ABB RobotStudio station: Laboratorio_simula.rspag

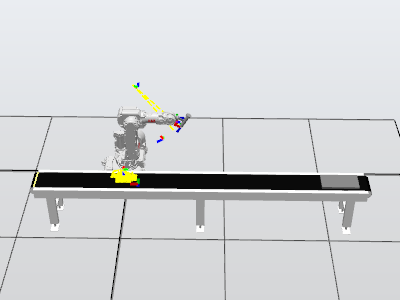
--- station ---
Station Project2 (saved by RobotStudio 25.3.11371.0)
Controller IRB140_6_81
  mechanical unit ROB_1: IRB140_6_81_C_03, 6 joints, base frame (0, 0, 0) mm
Layout (positions relative to the parent item):
  - IRB140_6_81_C_03 [mechanism, from %ABB.RobotStudio.Models.IRB140%\IRB140_6_81_C_G_03.rslib] at (0, 0, 0) mm; joint values [0, 0, 0, 0, 0, 0] (rad or m)
  - Soporte_final [mechanism] at (515, 0, 712) mm, rotated rx 0 ry 90 rz 0 deg
      TCP Soporte_final at (-0.03, 41.69, 114.81) mm, rotated rx 0 ry 30 rz -90 deg
      links: Soporte_7
  - Part_1 [part] at (-100, -130, -23) mm, size 280 x 180 x 80 mm
  - Rutina_Banda [smart component]
      signals: DI Activar_banda
      connections:
        Rutina_Banda.DI_01 -> PhysicsControl.SurfaceVelocityEnabled
        LineSensor_2.SensorOut -> Source.Execute
        Rutina_Banda.Activar_banda -> PhysicsControl.SurfaceVelocityEnabled
    - PhysicsControl [smart component, from Components\PhysicsControl.rslib]
        properties: Object=Belt Conveyor; Behavior=1; SurfaceVelocity=0.2
    - Belt Conveyor [part], size 3227.3 x 408.1 x 489.7 mm
    - Part_2 [part] at (2075.83, -708.5, 486.6) mm, size 350 x 180 x 20 mm
    - Source [smart component, from Components\Source.rslib]
        properties: Source=Part_2; Copy=(none); Parent=(none); Position=[2.079365 -0.71 0.517]; Orientation=[0 0 0]; Transient=true; PhysicsBehavior=-1
    - LineSensor_2 [smart component, from Components\LineSensor.rslib]
        properties: Start=[-0.8 -0.82 0.487]; End=[-0.8 -0.6 0.487]; Length=0.22; Radius=0.00152284263959391; Tag=(none); SenseMultiple=false; SensedPart=(none); SensedPoint=[0 0 0]
      - _sensorPart_ [part], size 3 x 220 x 3 mm
Attachment: Soporte_final is attached to IRB140_6_81_C_03 / Link6
Station logic (signal -> signal, property => property):
  IRB140_6_81.Conveyor_INV -> Rutina_Banda.Activar_banda

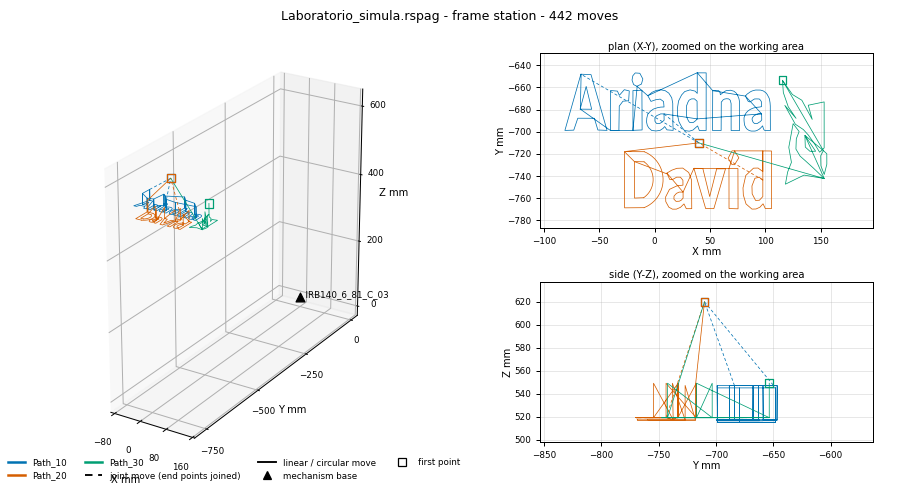
[picture p0: tool path of Laboratorio_simula.rspag in frame station, 442 of 446 moves have a stored position in this frame; points joined in program order, loops and branches not executed]
--- Controller Data/IRB140_6_81/RAPID/TASK1/PROGMOD/CalibData.mod ---
MODULE CalibData
ENDMODULE

--- Controller Data/IRB140_6_81/RAPID/TASK1/PROGMOD/Module3.mod ---
MODULE Module3
    CONST robtarget Target_200:=[[246.278,151.897,-25],[0.707106781,0,0,0.707106781],[-1,0,-1,1],[9E+09,9E+09,9E+09,9E+09,9E+09,9E+09]];
    CONST robtarget Target_210:=[[246.513,151.995,5],[0.707106781,0,0,0.707106781],[-1,0,-1,1],[9E+09,9E+09,9E+09,9E+09,9E+09,9E+09]];
    CONST robtarget Target_220:=[[237.364,151.636,5],[0.707106781,0,0,0.707106781],[-1,0,-1,1],[9E+09,9E+09,9E+09,9E+09,9E+09,9E+09]];
    CONST robtarget Target_230:=[[222.871,101.286,5],[0.707106781,0,0,0.707106781],[-1,0,-1,1],[9E+09,9E+09,9E+09,9E+09,9E+09,9E+09]];
    CONST robtarget Target_240:=[[231.165,101.624,5],[0.707106781,0,0,0.707106781],[-1,0,-1,1],[9E+09,9E+09,9E+09,9E+09,9E+09,9E+09]];
    CONST robtarget Target_250:=[[234.333,112.207,5],[0.707106781,0,0,0.707106781],[-1,0,-1,1],[9E+09,9E+09,9E+09,9E+09,9E+09,9E+09]];
    CONST robtarget Target_260:=[[249.288,112.26,5],[0.707106781,0,0,0.707106781],[-1,0,-1,1],[9E+09,9E+09,9E+09,9E+09,9E+09,9E+09]];
    CONST robtarget Target_270:=[[252.931,101.499,5],[0.707106781,0,0,0.707106781],[-1,0,-1,1],[9E+09,9E+09,9E+09,9E+09,9E+09,9E+09]];
    CONST robtarget Target_280:=[[260.918,101.25,5],[0.707106781,0,0,0.707106781],[-1,0,-1,1],[9E+09,9E+09,9E+09,9E+09,9E+09,9E+09]];
    CONST robtarget Target_290:=[[246.984,120.449,-25],[0.707106781,0,0,0.707106781],[-1,0,-1,1],[9E+09,9E+09,9E+09,9E+09,9E+09,9E+09]];
    CONST robtarget Target_300:=[[247.166,120.45,5],[0.707106781,0,0,0.707106781],[-1,0,-1,1],[9E+09,9E+09,9E+09,9E+09,9E+09,9E+09]];
    CONST robtarget Target_310:=[[236.764,120.36,5],[0.707106781,0,0,0.707106781],[-1,0,-1,1],[9E+09,9E+09,9E+09,9E+09,9E+09,9E+09]];
    CONST robtarget Target_320:=[[241.731,140.965,5],[0.707106781,0,0,0.707106781],[-1,0,-1,1],[9E+09,9E+09,9E+09,9E+09,9E+09,9E+09]];
    CONST robtarget Target_330:=[[219.929,101.246,-25],[0.707106781,0,0,0.707106781],[-1,0,-1,1],[9E+09,9E+09,9E+09,9E+09,9E+09,9E+09]];
    CONST robtarget Target_340:=[[219.745,101.297,5],[0.707106781,0,0,0.707106781],[-1,0,-1,1],[9E+09,9E+09,9E+09,9E+09,9E+09,9E+09]];
    CONST robtarget Target_350:=[[212.197,101.132,5],[0.707106781,0,0,0.707106781],[-1,0,-1,1],[9E+09,9E+09,9E+09,9E+09,9E+09,9E+09]];
    CONST robtarget Target_360:=[[211.858,123.214,5],[0.707106781,0,0,0.707106781],[-1,0,-1,1],[9E+09,9E+09,9E+09,9E+09,9E+09,9E+09]];
    CONST robtarget Target_370:=[[208.528,127.633,5],[0.707106781,0,0,0.707106781],[-1,0,-1,1],[9E+09,9E+09,9E+09,9E+09,9E+09,9E+09]];
    CONST robtarget Target_380:=[[203.388,128.012,5],[0.707106781,0,0,0.707106781],[-1,0,-1,1],[9E+09,9E+09,9E+09,9E+09,9E+09,9E+09]];
    CONST robtarget Target_390:=[[202.821,136.911,5],[0.707106781,0,0,0.707106781],[-1,0,-1,1],[9E+09,9E+09,9E+09,9E+09,9E+09,9E+09]];
    CONST robtarget Target_400:=[[207.318,137.995,5],[0.707106781,0,0,0.707106781],[-1,0,-1,1],[9E+09,9E+09,9E+09,9E+09,9E+09,9E+09]];
    CONST robtarget Target_410:=[[211.798,132.906,5],[0.707106781,0,0,0.707106781],[-1,0,-1,1],[9E+09,9E+09,9E+09,9E+09,9E+09,9E+09]];
    CONST robtarget Target_420:=[[213.511,136.735,5],[0.707106781,0,0,0.707106781],[-1,0,-1,1],[9E+09,9E+09,9E+09,9E+09,9E+09,9E+09]];
    CONST robtarget Target_430:=[[219.776,137.262,5],[0.707106781,0,0,0.707106781],[-1,0,-1,1],[9E+09,9E+09,9E+09,9E+09,9E+09,9E+09]];
    CONST robtarget Target_440:=[[219.929,116.68,5],[0.707106781,0,0,0.707106781],[-1,0,-1,1],[9E+09,9E+09,9E+09,9E+09,9E+09,9E+09]];
    CONST robtarget Target_450:=[[199.531,101.071,-27],[0.707106781,0,0,0.707106781],[-1,0,-1,1],[9E+09,9E+09,9E+09,9E+09,9E+09,9E+09]];
    CONST robtarget Target_460:=[[199.496,101.319,3],[0.707106781,0,0,0.707106781],[-1,0,-1,1],[9E+09,9E+09,9E+09,9E+09,9E+09,9E+09]];
    CONST robtarget Target_470:=[[199.502,137.231,3],[0.707106781,0,0,0.707106781],[-1,0,-1,1],[9E+09,9E+09,9E+09,9E+09,9E+09,9E+09]];
    CONST robtarget Target_480:=[[191.425,137.513,3],[0.707106781,0,0,0.707106781],[-1,0,-1,1],[9E+09,9E+09,9E+09,9E+09,9E+09,9E+09]];
    CONST robtarget Target_490:=[[191.227,101.671,3],[0.707106781,0,0,0.707106781],[-1,0,-1,1],[9E+09,9E+09,9E+09,9E+09,9E+09,9E+09]];
    CONST robtarget Target_500:=[[195.697,140.971,-27],[0.707106781,0,0,0.707106781],[-1,0,-1,1],[9E+09,9E+09,9E+09,9E+09,9E+09,9E+09]];
    CONST robtarget Target_510:=[[195.891,141.123,3],[0.707106781,0,0,0.707106781],[-1,0,-1,1],[9E+09,9E+09,9E+09,9E+09,9E+09,9E+09]];
    CONST robtarget Target_520:=[[191.844,143.083,3],[0.707106781,0,0,0.707106781],[-1,0,-1,1],[9E+09,9E+09,9E+09,9E+09,9E+09,9E+09]];
    CONST robtarget Target_530:=[[190.566,147.695,3],[0.707106781,0,0,0.707106781],[-1,0,-1,1],[9E+09,9E+09,9E+09,9E+09,9E+09,9E+09]];
    CONST robtarget Target_540:=[[193.297,152.839,3],[0.707106781,0,0,0.707106781],[-1,0,-1,1],[9E+09,9E+09,9E+09,9E+09,9E+09,9E+09]];
    CONST robtarget Target_550:=[[197.437,153.127,3],[0.707106781,0,0,0.707106781],[-1,0,-1,1],[9E+09,9E+09,9E+09,9E+09,9E+09,9E+09]];
    CONST robtarget Target_560:=[[199.597,150.616,3],[0.707106781,0,0,0.707106781],[-1,0,-1,1],[9E+09,9E+09,9E+09,9E+09,9E+09,9E+09]];
    CONST robtarget Target_570:=[[200.339,146.707,3],[0.707106781,0,0,0.707106781],[-1,0,-1,1],[9E+09,9E+09,9E+09,9E+09,9E+09,9E+09]];
    CONST robtarget Target_580:=[[198.927,142.651,3],[0.707106781,0,0,0.707106781],[-1,0,-1,1],[9E+09,9E+09,9E+09,9E+09,9E+09,9E+09]];
    CONST robtarget Target_590:=[[196.108,141.187,3],[0.707106781,0,0,0.707106781],[-1,0,-1,1],[9E+09,9E+09,9E+09,9E+09,9E+09,9E+09]];
    CONST robtarget Target_600:=[[185.991,132.618,-27],[0.707106781,0,0,0.707106781],[-1,0,-1,1],[9E+09,9E+09,9E+09,9E+09,9E+09,9E+09]];
    CONST robtarget Target_610:=[[186.042,132.532,3],[0.707106781,0,0,0.707106781],[-1,0,-1,1],[9E+09,9E+09,9E+09,9E+09,9E+09,9E+09]];
    CONST robtarget Target_620:=[[183.25,127.438,3],[0.707106781,0,0,0.707106781],[-1,0,-1,1],[9E+09,9E+09,9E+09,9E+09,9E+09,9E+09]];
    CONST robtarget Target_630:=[[179.02,128.919,3],[0.707106781,0,0,0.707106781],[-1,0,-1,1],[9E+09,9E+09,9E+09,9E+09,9E+09,9E+09]];
    CONST robtarget Target_640:=[[174.917,129.535,3],[0.707106781,0,0,0.707106781],[-1,0,-1,1],[9E+09,9E+09,9E+09,9E+09,9E+09,9E+09]];
    CONST robtarget Target_650:=[[171.888,127.333,3],[0.707106781,0,0,0.707106781],[-1,0,-1,1],[9E+09,9E+09,9E+09,9E+09,9E+09,9E+09]];
    CONST robtarget Target_660:=[[171.44,122.412,3],[0.707106781,0,0,0.707106781],[-1,0,-1,1],[9E+09,9E+09,9E+09,9E+09,9E+09,9E+09]];
    CONST robtarget Target_670:=[[174.411,122.301,3],[0.707106781,0,0,0.707106781],[-1,0,-1,1],[9E+09,9E+09,9E+09,9E+09,9E+09,9E+09]];
    CONST robtarget Target_680:=[[177.393,121.743,3],[0.707106781,0,0,0.707106781],[-1,0,-1,1],[9E+09,9E+09,9E+09,9E+09,9E+09,9E+09]];
    CONST robtarget Target_690:=[[181.014,120.522,3],[0.707106781,0,0,0.707106781],[-1,0,-1,1],[9E+09,9E+09,9E+09,9E+09,9E+09,9E+09]];
    CONST robtarget Target_700:=[[183.834,118.516,3],[0.707106781,0,0,0.707106781],[-1,0,-1,1],[9E+09,9E+09,9E+09,9E+09,9E+09,9E+09]];
    CONST robtarget Target_710:=[[186.198,115.714,3],[0.707106781,0,0,0.707106781],[-1,0,-1,1],[9E+09,9E+09,9E+09,9E+09,9E+09,9E+09]];
    CONST robtarget Target_720:=[[187.033,112.205,3],[0.707106781,0,0,0.707106781],[-1,0,-1,1],[9E+09,9E+09,9E+09,9E+09,9E+09,9E+09]];
    CONST robtarget Target_730:=[[187.201,108.775,3],[0.707106781,0,0,0.707106781],[-1,0,-1,1],[9E+09,9E+09,9E+09,9E+09,9E+09,9E+09]];
    CONST robtarget Target_740:=[[186.537,105.714,3],[0.707106781,0,0,0.707106781],[-1,0,-1,1],[9E+09,9E+09,9E+09,9E+09,9E+09,9E+09]];
    CONST robtarget Target_750:=[[185.137,103.46,3],[0.707106781,0,0,0.707106781],[-1,0,-1,1],[9E+09,9E+09,9E+09,9E+09,9E+09,9E+09]];
    CONST robtarget Target_760:=[[182.665,101.233,3],[0.707106781,0,0,0.707106781],[-1,0,-1,1],[9E+09,9E+09,9E+09,9E+09,9E+09,9E+09]];
    CONST robtarget Target_770:=[[178.705,100.766,3],[0.707106781,0,0,0.707106781],[-1,0,-1,1],[9E+09,9E+09,9E+09,9E+09,9E+09,9E+09]];
    CONST robtarget Target_780:=[[175.006,101.312,3],[0.707106781,0,0,0.707106781],[-1,0,-1,1],[9E+09,9E+09,9E+09,9E+09,9E+09,9E+09]];
    CONST robtarget Target_790:=[[172.351,103.047,3],[0.707106781,0,0,0.707106781],[-1,0,-1,1],[9E+09,9E+09,9E+09,9E+09,9E+09,9E+09]];
    CONST robtarget Target_800:=[[170.872,104.731,3],[0.707106781,0,0,0.707106781],[-1,0,-1,1],[9E+09,9E+09,9E+09,9E+09,9E+09,9E+09]];
    CONST robtarget Target_810:=[[168.786,101.751,3],[0.707106781,0,0,0.707106781],[-1,0,-1,1],[9E+09,9E+09,9E+09,9E+09,9E+09,9E+09]];
    CONST robtarget Target_820:=[[163.181,101.281,3],[0.707106781,0,0,0.707106781],[-1,0,-1,1],[9E+09,9E+09,9E+09,9E+09,9E+09,9E+09]];
    CONST robtarget Target_830:=[[163.458,107.365,3],[0.707106781,0,0,0.707106781],[-1,0,-1,1],[9E+09,9E+09,9E+09,9E+09,9E+09,9E+09]];
    CONST robtarget Target_840:=[[163.573,125.763,3],[0.707106781,0,0,0.707106781],[-1,0,-1,1],[9E+09,9E+09,9E+09,9E+09,9E+09,9E+09]];
    CONST robtarget Target_850:=[[164.518,130.704,3],[0.707106781,0,0,0.707106781],[-1,0,-1,1],[9E+09,9E+09,9E+09,9E+09,9E+09,9E+09]];
    CONST robtarget Target_860:=[[167.119,134.898,3],[0.707106781,0,0,0.707106781],[-1,0,-1,1],[9E+09,9E+09,9E+09,9E+09,9E+09,9E+09]];
    CONST robtarget Target_870:=[[170.356,137.106,3],[0.707106781,0,0,0.707106781],[-1,0,-1,1],[9E+09,9E+09,9E+09,9E+09,9E+09,9E+09]];
    CONST robtarget Target_880:=[[174.256,137.887,3],[0.707106781,0,0,0.707106781],[-1,0,-1,1],[9E+09,9E+09,9E+09,9E+09,9E+09,9E+09]];
    CONST robtarget Target_890:=[[178.229,137.441,3],[0.707106781,0,0,0.707106781],[-1,0,-1,1],[9E+09,9E+09,9E+09,9E+09,9E+09,9E+09]];
    CONST robtarget Target_900:=[[182.159,135.699,3],[0.707106781,0,0,0.707106781],[-1,0,-1,1],[9E+09,9E+09,9E+09,9E+09,9E+09,9E+09]];
    CONST robtarget Target_910:=[[141.477,153.34,-27],[0.707106781,0,0,0.707106781],[-1,0,-1,1],[9E+09,9E+09,9E+09,9E+09,9E+09,9E+09]];
    CONST robtarget Target_920:=[[141.463,153.223,3],[0.707106781,0,0,0.707106781],[-1,0,-1,1],[9E+09,9E+09,9E+09,9E+09,9E+09,9E+09]];
    CONST robtarget Target_930:=[[133.41,153.195,3],[0.707106781,0,0,0.707106781],[-1,0,-1,1],[9E+09,9E+09,9E+09,9E+09,9E+09,9E+09]];
    CONST robtarget Target_940:=[[133.441,101.226,3],[0.707106781,0,0,0.707106781],[-1,0,-1,1],[9E+09,9E+09,9E+09,9E+09,9E+09,9E+09]];
    CONST robtarget Target_950:=[[139.552,101.121,3],[0.707106781,0,0,0.707106781],[-1,0,-1,1],[9E+09,9E+09,9E+09,9E+09,9E+09,9E+09]];
    CONST robtarget Target_960:=[[141.139,105.303,3],[0.707106781,0,0,0.707106781],[-1,0,-1,1],[9E+09,9E+09,9E+09,9E+09,9E+09,9E+09]];
    CONST robtarget Target_970:=[[142.695,103.897,3],[0.707106781,0,0,0.707106781],[-1,0,-1,1],[9E+09,9E+09,9E+09,9E+09,9E+09,9E+09]];
    CONST robtarget Target_980:=[[145.383,101.548,3],[0.707106781,0,0,0.707106781],[-1,0,-1,1],[9E+09,9E+09,9E+09,9E+09,9E+09,9E+09]];
    CONST robtarget Target_990:=[[148.713,100.557,3],[0.707106781,0,0,0.707106781],[-1,0,-1,1],[9E+09,9E+09,9E+09,9E+09,9E+09,9E+09]];
    CONST robtarget Target_1000:=[[153.006,101.152,3],[0.707106781,0,0,0.707106781],[-1,0,-1,1],[9E+09,9E+09,9E+09,9E+09,9E+09,9E+09]];
    CONST robtarget Target_1010:=[[155.494,104.348,3],[0.707106781,0,0,0.707106781],[-1,0,-1,1],[9E+09,9E+09,9E+09,9E+09,9E+09,9E+09]];
    CONST robtarget Target_1020:=[[157.99,109.125,3],[0.707106781,0,0,0.707106781],[-1,0,-1,1],[9E+09,9E+09,9E+09,9E+09,9E+09,9E+09]];
    CONST robtarget Target_1030:=[[159.201,114.82,3],[0.707106781,0,0,0.707106781],[-1,0,-1,1],[9E+09,9E+09,9E+09,9E+09,9E+09,9E+09]];
    CONST robtarget Target_1040:=[[159.416,120.79,3],[0.707106781,0,0,0.707106781],[-1,0,-1,1],[9E+09,9E+09,9E+09,9E+09,9E+09,9E+09]];
    CONST robtarget Target_1050:=[[158.345,127.799,3],[0.707106781,0,0,0.707106781],[-1,0,-1,1],[9E+09,9E+09,9E+09,9E+09,9E+09,9E+09]];
    CONST robtarget Target_1060:=[[155.578,133.274,3],[0.707106781,0,0,0.707106781],[-1,0,-1,1],[9E+09,9E+09,9E+09,9E+09,9E+09,9E+09]];
    CONST robtarget Target_1070:=[[152.755,136.341,3],[0.707106781,0,0,0.707106781],[-1,0,-1,1],[9E+09,9E+09,9E+09,9E+09,9E+09,9E+09]];
    CONST robtarget Target_1080:=[[147.939,137.836,3],[0.707106781,0,0,0.707106781],[-1,0,-1,1],[9E+09,9E+09,9E+09,9E+09,9E+09,9E+09]];
    CONST robtarget Target_1090:=[[143.364,136.708,3],[0.707106781,0,0,0.707106781],[-1,0,-1,1],[9E+09,9E+09,9E+09,9E+09,9E+09,9E+09]];
    CONST robtarget Target_1100:=[[141.46,134.647,3],[0.707106781,0,0,0.707106781],[-1,0,-1,1],[9E+09,9E+09,9E+09,9E+09,9E+09,9E+09]];
    CONST robtarget Target_1110:=[[127.462,137.098,-27],[0.707106781,0,0,0.707106781],[-1,0,-1,1],[9E+09,9E+09,9E+09,9E+09,9E+09,9E+09]];
    CONST robtarget Target_1120:=[[127.513,137.169,3],[0.707106781,0,0,0.707106781],[-1,0,-1,1],[9E+09,9E+09,9E+09,9E+09,9E+09,9E+09]];
    CONST robtarget Target_1130:=[[122.089,137.155,3],[0.707106781,0,0,0.707106781],[-1,0,-1,1],[9E+09,9E+09,9E+09,9E+09,9E+09,9E+09]];
    CONST robtarget Target_1140:=[[120.939,135.863,3],[0.707106781,0,0,0.707106781],[-1,0,-1,1],[9E+09,9E+09,9E+09,9E+09,9E+09,9E+09]];
    CONST robtarget Target_1150:=[[120.597,133.446,3],[0.707106781,0,0,0.707106781],[-1,0,-1,1],[9E+09,9E+09,9E+09,9E+09,9E+09,9E+09]];
    CONST robtarget Target_1160:=[[118.764,134.854,3],[0.707106781,0,0,0.707106781],[-1,0,-1,1],[9E+09,9E+09,9E+09,9E+09,9E+09,9E+09]];
    CONST robtarget Target_1170:=[[117.354,136.062,3],[0.707106781,0,0,0.707106781],[-1,0,-1,1],[9E+09,9E+09,9E+09,9E+09,9E+09,9E+09]];
    CONST robtarget Target_1180:=[[115.44,137.119,3],[0.707106781,0,0,0.707106781],[-1,0,-1,1],[9E+09,9E+09,9E+09,9E+09,9E+09,9E+09]];
    CONST robtarget Target_1190:=[[111.466,137.53,3],[0.707106781,0,0,0.707106781],[-1,0,-1,1],[9E+09,9E+09,9E+09,9E+09,9E+09,9E+09]];
    CONST robtarget Target_1200:=[[108.302,136.627,3],[0.707106781,0,0,0.707106781],[-1,0,-1,1],[9E+09,9E+09,9E+09,9E+09,9E+09,9E+09]];
    CONST robtarget Target_1210:=[[106.188,134.824,3],[0.707106781,0,0,0.707106781],[-1,0,-1,1],[9E+09,9E+09,9E+09,9E+09,9E+09,9E+09]];
    CONST robtarget Target_1220:=[[104.697,132.135,3],[0.707106781,0,0,0.707106781],[-1,0,-1,1],[9E+09,9E+09,9E+09,9E+09,9E+09,9E+09]];
    CONST robtarget Target_1230:=[[103.786,129.731,3],[0.707106781,0,0,0.707106781],[-1,0,-1,1],[9E+09,9E+09,9E+09,9E+09,9E+09,9E+09]];
    CONST robtarget Target_1240:=[[103.252,126.813,3],[0.707106781,0,0,0.707106781],[-1,0,-1,1],[9E+09,9E+09,9E+09,9E+09,9E+09,9E+09]];
    CONST robtarget Target_1250:=[[103.231,101.169,3],[0.707106781,0,0,0.707106781],[-1,0,-1,1],[9E+09,9E+09,9E+09,9E+09,9E+09,9E+09]];
    CONST robtarget Target_1260:=[[110.877,101.137,3],[0.707106781,0,0,0.707106781],[-1,0,-1,1],[9E+09,9E+09,9E+09,9E+09,9E+09,9E+09]];
    CONST robtarget Target_1270:=[[110.901,125.483,3],[0.707106781,0,0,0.707106781],[-1,0,-1,1],[9E+09,9E+09,9E+09,9E+09,9E+09,9E+09]];
    CONST robtarget Target_1280:=[[111.711,128.545,3],[0.707106781,0,0,0.707106781],[-1,0,-1,1],[9E+09,9E+09,9E+09,9E+09,9E+09,9E+09]];
    CONST robtarget Target_1290:=[[113.108,129.695,3],[0.707106781,0,0,0.707106781],[-1,0,-1,1],[9E+09,9E+09,9E+09,9E+09,9E+09,9E+09]];
    CONST robtarget Target_1300:=[[115.021,129.869,3],[0.707106781,0,0,0.707106781],[-1,0,-1,1],[9E+09,9E+09,9E+09,9E+09,9E+09,9E+09]];
    CONST robtarget Target_1310:=[[116.884,129.541,3],[0.707106781,0,0,0.707106781],[-1,0,-1,1],[9E+09,9E+09,9E+09,9E+09,9E+09,9E+09]];
    CONST robtarget Target_1320:=[[118.097,128.875,3],[0.707106781,0,0,0.707106781],[-1,0,-1,1],[9E+09,9E+09,9E+09,9E+09,9E+09,9E+09]];
    CONST robtarget Target_1330:=[[118.947,127.721,3],[0.707106781,0,0,0.707106781],[-1,0,-1,1],[9E+09,9E+09,9E+09,9E+09,9E+09,9E+09]];
    CONST robtarget Target_1340:=[[119.769,126.854,3],[0.707106781,0,0,0.707106781],[-1,0,-1,1],[9E+09,9E+09,9E+09,9E+09,9E+09,9E+09]];
    CONST robtarget Target_1350:=[[119.905,101.166,3],[0.707106781,0,0,0.707106781],[-1,0,-1,1],[9E+09,9E+09,9E+09,9E+09,9E+09,9E+09]];
    CONST robtarget Target_1360:=[[127.655,101.147,3],[0.707106781,0,0,0.707106781],[-1,0,-1,1],[9E+09,9E+09,9E+09,9E+09,9E+09,9E+09]];
    CONST robtarget Target_1370:=[[98.011,132.261,-27],[0.707106781,0,0,0.707106781],[-1,0,-1,1],[9E+09,9E+09,9E+09,9E+09,9E+09,9E+09]];
    CONST robtarget Target_1380:=[[97.987,132.237,3],[0.707106781,0,0,0.707106781],[-1,0,-1,1],[9E+09,9E+09,9E+09,9E+09,9E+09,9E+09]];
    CONST robtarget Target_1390:=[[95.469,127.492,3],[0.707106781,0,0,0.707106781],[-1,0,-1,1],[9E+09,9E+09,9E+09,9E+09,9E+09,9E+09]];
    CONST robtarget Target_1400:=[[94.177,127.002,3],[0.707106781,0,0,0.707106781],[-1,0,-1,1],[9E+09,9E+09,9E+09,9E+09,9E+09,9E+09]];
    CONST robtarget Target_1410:=[[93.07,127.439,3],[0.707106781,0,0,0.707106781],[-1,0,-1,1],[9E+09,9E+09,9E+09,9E+09,9E+09,9E+09]];
    CONST robtarget Target_1420:=[[91.226,128.754,3],[0.707106781,0,0,0.707106781],[-1,0,-1,1],[9E+09,9E+09,9E+09,9E+09,9E+09,9E+09]];
    CONST robtarget Target_1430:=[[89.761,129.648,3],[0.707106781,0,0,0.707106781],[-1,0,-1,1],[9E+09,9E+09,9E+09,9E+09,9E+09,9E+09]];
    CONST robtarget Target_1440:=[[87.721,129.697,3],[0.707106781,0,0,0.707106781],[-1,0,-1,1],[9E+09,9E+09,9E+09,9E+09,9E+09,9E+09]];
    CONST robtarget Target_1450:=[[85.497,129.633,3],[0.707106781,0,0,0.707106781],[-1,0,-1,1],[9E+09,9E+09,9E+09,9E+09,9E+09,9E+09]];
    CONST robtarget Target_1460:=[[84.322,128.462,3],[0.707106781,0,0,0.707106781],[-1,0,-1,1],[9E+09,9E+09,9E+09,9E+09,9E+09,9E+09]];
    CONST robtarget Target_1470:=[[83.511,127.021,3],[0.707106781,0,0,0.707106781],[-1,0,-1,1],[9E+09,9E+09,9E+09,9E+09,9E+09,9E+09]];
    CONST robtarget Target_1480:=[[83.433,124.649,3],[0.707106781,0,0,0.707106781],[-1,0,-1,1],[9E+09,9E+09,9E+09,9E+09,9E+09,9E+09]];
    CONST robtarget Target_1490:=[[83.449,122.703,3],[0.707106781,0,0,0.707106781],[-1,0,-1,1],[9E+09,9E+09,9E+09,9E+09,9E+09,9E+09]];
    CONST robtarget Target_1500:=[[85.232,122.344,3],[0.707106781,0,0,0.707106781],[-1,0,-1,1],[9E+09,9E+09,9E+09,9E+09,9E+09,9E+09]];
    CONST robtarget Target_1510:=[[87.719,122.088,3],[0.707106781,0,0,0.707106781],[-1,0,-1,1],[9E+09,9E+09,9E+09,9E+09,9E+09,9E+09]];
    CONST robtarget Target_1520:=[[90.166,121.644,3],[0.707106781,0,0,0.707106781],[-1,0,-1,1],[9E+09,9E+09,9E+09,9E+09,9E+09,9E+09]];
    CONST robtarget Target_1530:=[[91.454,121.192,3],[0.707106781,0,0,0.707106781],[-1,0,-1,1],[9E+09,9E+09,9E+09,9E+09,9E+09,9E+09]];
    CONST robtarget Target_1540:=[[92.626,120.652,3],[0.707106781,0,0,0.707106781],[-1,0,-1,1],[9E+09,9E+09,9E+09,9E+09,9E+09,9E+09]];
    CONST robtarget Target_1550:=[[93.765,120.146,3],[0.707106781,0,0,0.707106781],[-1,0,-1,1],[9E+09,9E+09,9E+09,9E+09,9E+09,9E+09]];
    CONST robtarget Target_1560:=[[94.487,119.64,3],[0.707106781,0,0,0.707106781],[-1,0,-1,1],[9E+09,9E+09,9E+09,9E+09,9E+09,9E+09]];
    CONST robtarget Target_1570:=[[95.219,119.089,3],[0.707106781,0,0,0.707106781],[-1,0,-1,1],[9E+09,9E+09,9E+09,9E+09,9E+09,9E+09]];
    CONST robtarget Target_1580:=[[95.865,118.666,3],[0.707106781,0,0,0.707106781],[-1,0,-1,1],[9E+09,9E+09,9E+09,9E+09,9E+09,9E+09]];
    CONST robtarget Target_1590:=[[96.271,118.099,3],[0.707106781,0,0,0.707106781],[-1,0,-1,1],[9E+09,9E+09,9E+09,9E+09,9E+09,9E+09]];
    CONST robtarget Target_1600:=[[96.723,117.792,3],[0.707106781,0,0,0.707106781],[-1,0,-1,1],[9E+09,9E+09,9E+09,9E+09,9E+09,9E+09]];
    CONST robtarget Target_1610:=[[97.248,117.224,3],[0.707106781,0,0,0.707106781],[-1,0,-1,1],[9E+09,9E+09,9E+09,9E+09,9E+09,9E+09]];
    CONST robtarget Target_1620:=[[97.549,116.742,3],[0.707106781,0,0,0.707106781],[-1,0,-1,1],[9E+09,9E+09,9E+09,9E+09,9E+09,9E+09]];
    CONST robtarget Target_1630:=[[97.955,116.258,3],[0.707106781,0,0,0.707106781],[-1,0,-1,1],[9E+09,9E+09,9E+09,9E+09,9E+09,9E+09]];
    CONST robtarget Target_1640:=[[98.251,115.523,3],[0.707106781,0,0,0.707106781],[-1,0,-1,1],[9E+09,9E+09,9E+09,9E+09,9E+09,9E+09]];
    CONST robtarget Target_1650:=[[98.546,114.76,3],[0.707106781,0,0,0.707106781],[-1,0,-1,1],[9E+09,9E+09,9E+09,9E+09,9E+09,9E+09]];
    CONST robtarget Target_1660:=[[98.886,113.804,3],[0.707106781,0,0,0.707106781],[-1,0,-1,1],[9E+09,9E+09,9E+09,9E+09,9E+09,9E+09]];
    CONST robtarget Target_1670:=[[99.236,112.637,3],[0.707106781,0,0,0.707106781],[-1,0,-1,1],[9E+09,9E+09,9E+09,9E+09,9E+09,9E+09]];
    CONST robtarget Target_1680:=[[99.219,109.938,3],[0.707106781,0,0,0.707106781],[-1,0,-1,1],[9E+09,9E+09,9E+09,9E+09,9E+09,9E+09]];
    CONST robtarget Target_1690:=[[99.02,108.205,3],[0.707106781,0,0,0.707106781],[-1,0,-1,1],[9E+09,9E+09,9E+09,9E+09,9E+09,9E+09]];
    CONST robtarget Target_1700:=[[98.851,106.622,3],[0.707106781,0,0,0.707106781],[-1,0,-1,1],[9E+09,9E+09,9E+09,9E+09,9E+09,9E+09]];
    CONST robtarget Target_1710:=[[98.527,105.563,3],[0.707106781,0,0,0.707106781],[-1,0,-1,1],[9E+09,9E+09,9E+09,9E+09,9E+09,9E+09]];
    CONST robtarget Target_1720:=[[98.139,104.962,3],[0.707106781,0,0,0.707106781],[-1,0,-1,1],[9E+09,9E+09,9E+09,9E+09,9E+09,9E+09]];
    CONST robtarget Target_1730:=[[97.776,104.049,3],[0.707106781,0,0,0.707106781],[-1,0,-1,1],[9E+09,9E+09,9E+09,9E+09,9E+09,9E+09]];
    CONST robtarget Target_1740:=[[97.409,103.55,3],[0.707106781,0,0,0.707106781],[-1,0,-1,1],[9E+09,9E+09,9E+09,9E+09,9E+09,9E+09]];
    CONST robtarget Target_1750:=[[97.069,103.049,3],[0.707106781,0,0,0.707106781],[-1,0,-1,1],[9E+09,9E+09,9E+09,9E+09,9E+09,9E+09]];
    CONST robtarget Target_1760:=[[96.704,102.617,3],[0.707106781,0,0,0.707106781],[-1,0,-1,1],[9E+09,9E+09,9E+09,9E+09,9E+09,9E+09]];
    CONST robtarget Target_1770:=[[96.045,102.097,3],[0.707106781,0,0,0.707106781],[-1,0,-1,1],[9E+09,9E+09,9E+09,9E+09,9E+09,9E+09]];
    CONST robtarget Target_1780:=[[95.311,101.599,3],[0.707106781,0,0,0.707106781],[-1,0,-1,1],[9E+09,9E+09,9E+09,9E+09,9E+09,9E+09]];
    CONST robtarget Target_1790:=[[94.479,101.133,3],[0.707106781,0,0,0.707106781],[-1,0,-1,1],[9E+09,9E+09,9E+09,9E+09,9E+09,9E+09]];
    CONST robtarget Target_1800:=[[92.719,100.672,3],[0.707106781,0,0,0.707106781],[-1,0,-1,1],[9E+09,9E+09,9E+09,9E+09,9E+09,9E+09]];
    CONST robtarget Target_1810:=[[89.338,100.675,3],[0.707106781,0,0,0.707106781],[-1,0,-1,1],[9E+09,9E+09,9E+09,9E+09,9E+09,9E+09]];
    CONST robtarget Target_1820:=[[87.663,101.128,3],[0.707106781,0,0,0.707106781],[-1,0,-1,1],[9E+09,9E+09,9E+09,9E+09,9E+09,9E+09]];
    CONST robtarget Target_1830:=[[86.739,101.629,3],[0.707106781,0,0,0.707106781],[-1,0,-1,1],[9E+09,9E+09,9E+09,9E+09,9E+09,9E+09]];
    CONST robtarget Target_1840:=[[85.95,102.071,3],[0.707106781,0,0,0.707106781],[-1,0,-1,1],[9E+09,9E+09,9E+09,9E+09,9E+09,9E+09]];
    CONST robtarget Target_1850:=[[85.233,102.539,3],[0.707106781,0,0,0.707106781],[-1,0,-1,1],[9E+09,9E+09,9E+09,9E+09,9E+09,9E+09]];
    CONST robtarget Target_1860:=[[85.252,102.559,3],[0.707106781,0,0,0.707106781],[-1,0,-1,1],[9E+09,9E+09,9E+09,9E+09,9E+09,9E+09]];
    CONST robtarget Target_1870:=[[84.579,103.084,3],[0.707106781,0,0,0.707106781],[-1,0,-1,1],[9E+09,9E+09,9E+09,9E+09,9E+09,9E+09]];
    CONST robtarget Target_1880:=[[84.143,103.582,3],[0.707106781,0,0,0.707106781],[-1,0,-1,1],[9E+09,9E+09,9E+09,9E+09,9E+09,9E+09]];
    CONST robtarget Target_1890:=[[83.815,104.033,3],[0.707106781,0,0,0.707106781],[-1,0,-1,1],[9E+09,9E+09,9E+09,9E+09,9E+09,9E+09]];
    CONST robtarget Target_1900:=[[83.225,104.612,3],[0.707106781,0,0,0.707106781],[-1,0,-1,1],[9E+09,9E+09,9E+09,9E+09,9E+09,9E+09]];
    CONST robtarget Target_1910:=[[82.459,105.382,3],[0.707106781,0,0,0.707106781],[-1,0,-1,1],[9E+09,9E+09,9E+09,9E+09,9E+09,9E+09]];
    CONST robtarget Target_1920:=[[82.067,104.011,3],[0.707106781,0,0,0.707106781],[-1,0,-1,1],[9E+09,9E+09,9E+09,9E+09,9E+09,9E+09]];
    CONST robtarget Target_1930:=[[81.695,102.64,3],[0.707106781,0,0,0.707106781],[-1,0,-1,1],[9E+09,9E+09,9E+09,9E+09,9E+09,9E+09]];
    CONST robtarget Target_1940:=[[81.334,102.016,3],[0.707106781,0,0,0.707106781],[-1,0,-1,1],[9E+09,9E+09,9E+09,9E+09,9E+09,9E+09]];
    CONST robtarget Target_1950:=[[81.005,101.579,3],[0.707106781,0,0,0.707106781],[-1,0,-1,1],[9E+09,9E+09,9E+09,9E+09,9E+09,9E+09]];
    CONST robtarget Target_1960:=[[80.15,101.178,3],[0.707106781,0,0,0.707106781],[-1,0,-1,1],[9E+09,9E+09,9E+09,9E+09,9E+09,9E+09]];
    CONST robtarget Target_1970:=[[75.457,101.107,3],[0.707106781,0,0,0.707106781],[-1,0,-1,1],[9E+09,9E+09,9E+09,9E+09,9E+09,9E+09]];
    CONST robtarget Target_1980:=[[75.547,123.303,3],[0.707106781,0,0,0.707106781],[-1,0,-1,1],[9E+09,9E+09,9E+09,9E+09,9E+09,9E+09]];
    CONST robtarget Target_1990:=[[75.745,126.15,3],[0.707106781,0,0,0.707106781],[-1,0,-1,1],[9E+09,9E+09,9E+09,9E+09,9E+09,9E+09]];
    CONST robtarget Target_2000:=[[76.251,129.305,3],[0.707106781,0,0,0.707106781],[-1,0,-1,1],[9E+09,9E+09,9E+09,9E+09,9E+09,9E+09]];
    CONST robtarget Target_2010:=[[76.643,130.488,3],[0.707106781,0,0,0.707106781],[-1,0,-1,1],[9E+09,9E+09,9E+09,9E+09,9E+09,9E+09]];
    CONST robtarget Target_2020:=[[77.332,131.926,3],[0.707106781,0,0,0.707106781],[-1,0,-1,1],[9E+09,9E+09,9E+09,9E+09,9E+09,9E+09]];
    CONST robtarget Target_2030:=[[77.77,132.789,3],[0.707106781,0,0,0.707106781],[-1,0,-1,1],[9E+09,9E+09,9E+09,9E+09,9E+09,9E+09]];
    CONST robtarget Target_2040:=[[78.107,133.332,3],[0.707106781,0,0,0.707106781],[-1,0,-1,1],[9E+09,9E+09,9E+09,9E+09,9E+09,9E+09]];
    CONST robtarget Target_2050:=[[78.388,133.751,3],[0.707106781,0,0,0.707106781],[-1,0,-1,1],[9E+09,9E+09,9E+09,9E+09,9E+09,9E+09]];
    CONST robtarget Target_2060:=[[78.737,134.294,3],[0.707106781,0,0,0.707106781],[-1,0,-1,1],[9E+09,9E+09,9E+09,9E+09,9E+09,9E+09]];
    CONST robtarget Target_2070:=[[79.136,134.868,3],[0.707106781,0,0,0.707106781],[-1,0,-1,1],[9E+09,9E+09,9E+09,9E+09,9E+09,9E+09]];
    CONST robtarget Target_2080:=[[79.765,135.389,3],[0.707106781,0,0,0.707106781],[-1,0,-1,1],[9E+09,9E+09,9E+09,9E+09,9E+09,9E+09]];
    CONST robtarget Target_2090:=[[80.304,135.801,3],[0.707106781,0,0,0.707106781],[-1,0,-1,1],[9E+09,9E+09,9E+09,9E+09,9E+09,9E+09]];
    CONST robtarget Target_2100:=[[80.943,136.287,3],[0.707106781,0,0,0.707106781],[-1,0,-1,1],[9E+09,9E+09,9E+09,9E+09,9E+09,9E+09]];
    CONST robtarget Target_2110:=[[81.704,136.811,3],[0.707106781,0,0,0.707106781],[-1,0,-1,1],[9E+09,9E+09,9E+09,9E+09,9E+09,9E+09]];
    CONST robtarget Target_2120:=[[82.701,137.179,3],[0.707106781,0,0,0.707106781],[-1,0,-1,1],[9E+09,9E+09,9E+09,9E+09,9E+09,9E+09]];
    CONST robtarget Target_2130:=[[84.412,137.659,3],[0.707106781,0,0,0.707106781],[-1,0,-1,1],[9E+09,9E+09,9E+09,9E+09,9E+09,9E+09]];
    CONST robtarget Target_2140:=[[88.761,137.699,3],[0.707106781,0,0,0.707106781],[-1,0,-1,1],[9E+09,9E+09,9E+09,9E+09,9E+09,9E+09]];
    CONST robtarget Target_2150:=[[90.735,137.26,3],[0.707106781,0,0,0.707106781],[-1,0,-1,1],[9E+09,9E+09,9E+09,9E+09,9E+09,9E+09]];
    CONST robtarget Target_2160:=[[92.256,136.74,3],[0.707106781,0,0,0.707106781],[-1,0,-1,1],[9E+09,9E+09,9E+09,9E+09,9E+09,9E+09]];
    CONST robtarget Target_2170:=[[93.136,136.258,3],[0.707106781,0,0,0.707106781],[-1,0,-1,1],[9E+09,9E+09,9E+09,9E+09,9E+09,9E+09]];
    CONST robtarget Target_2180:=[[94.197,135.688,3],[0.707106781,0,0,0.707106781],[-1,0,-1,1],[9E+09,9E+09,9E+09,9E+09,9E+09,9E+09]];
    CONST robtarget Target_2190:=[[94.837,135.139,3],[0.707106781,0,0,0.707106781],[-1,0,-1,1],[9E+09,9E+09,9E+09,9E+09,9E+09,9E+09]];
    CONST robtarget Target_2200:=[[95.528,134.73,3],[0.707106781,0,0,0.707106781],[-1,0,-1,1],[9E+09,9E+09,9E+09,9E+09,9E+09,9E+09]];
    CONST robtarget Target_2210:=[[96.115,134.269,3],[0.707106781,0,0,0.707106781],[-1,0,-1,1],[9E+09,9E+09,9E+09,9E+09,9E+09,9E+09]];
    CONST robtarget Target_2220:=[[96.58,133.901,3],[0.707106781,0,0,0.707106781],[-1,0,-1,1],[9E+09,9E+09,9E+09,9E+09,9E+09,9E+09]];
    CONST robtarget Target_2230:=[[97.115,133.257,3],[0.707106781,0,0,0.707106781],[-1,0,-1,1],[9E+09,9E+09,9E+09,9E+09,9E+09,9E+09]];
    CONST robtarget Target_2240:=[[97.597,132.688,3],[0.707106781,0,0,0.707106781],[-1,0,-1,1],[9E+09,9E+09,9E+09,9E+09,9E+09,9E+09]];
    CONST robtarget Target_minihome:=[[140,90,-100],[0.707106781,0,0,0.707106781],[-1,0,-1,1],[9E+09,9E+09,9E+09,9E+09,9E+09,9E+09]];
    CONST robtarget Target_2250:=[[83.342,116.209,-27],[0.707106781,0,0,0.707106781],[-1,0,-1,1],[9E+09,9E+09,9E+09,9E+09,9E+09,9E+09]];
    CONST robtarget Target_2260:=[[83.357,116.248,3],[0.707106781,0,0,0.707106781],[-1,0,-1,1],[9E+09,9E+09,9E+09,9E+09,9E+09,9E+09]];
    CONST robtarget Target_2270:=[[83.249,110.742,3],[0.707106781,0,0,0.707106781],[-1,0,-1,1],[9E+09,9E+09,9E+09,9E+09,9E+09,9E+09]];
    CONST robtarget Target_2280:=[[83.528,110.403,3],[0.707106781,0,0,0.707106781],[-1,0,-1,1],[9E+09,9E+09,9E+09,9E+09,9E+09,9E+09]];
    CONST robtarget Target_2290:=[[83.916,109.924,3],[0.707106781,0,0,0.707106781],[-1,0,-1,1],[9E+09,9E+09,9E+09,9E+09,9E+09,9E+09]];
    CONST robtarget Target_2300:=[[84.293,109.456,3],[0.707106781,0,0,0.707106781],[-1,0,-1,1],[9E+09,9E+09,9E+09,9E+09,9E+09,9E+09]];
    CONST robtarget Target_2310:=[[84.94,108.951,3],[0.707106781,0,0,0.707106781],[-1,0,-1,1],[9E+09,9E+09,9E+09,9E+09,9E+09,9E+09]];
    CONST robtarget Target_2320:=[[85.814,108.513,3],[0.707106781,0,0,0.707106781],[-1,0,-1,1],[9E+09,9E+09,9E+09,9E+09,9E+09,9E+09]];
    CONST robtarget Target_2330:=[[141.495,111.664,-27],[0.707106781,0,0,0.707106781],[-1,0,-1,1],[9E+09,9E+09,9E+09,9E+09,9E+09,9E+09]];
    CONST robtarget Target_2340:=[[86.606,107.969,3],[0.707106781,0,0,0.707106781],[-1,0,-1,1],[9E+09,9E+09,9E+09,9E+09,9E+09,9E+09]];
    CONST robtarget Target_2350:=[[87.161,107.517,3],[0.707106781,0,0,0.707106781],[-1,0,-1,1],[9E+09,9E+09,9E+09,9E+09,9E+09,9E+09]];
    CONST robtarget Target_2360:=[[88.612,107.478,3],[0.707106781,0,0,0.707106781],[-1,0,-1,1],[9E+09,9E+09,9E+09,9E+09,9E+09,9E+09]];
    CONST robtarget Target_2370:=[[89.854,107.544,3],[0.707106781,0,0,0.707106781],[-1,0,-1,1],[9E+09,9E+09,9E+09,9E+09,9E+09,9E+09]];
    CONST robtarget Target_2380:=[[90.796,108.417,3],[0.707106781,0,0,0.707106781],[-1,0,-1,1],[9E+09,9E+09,9E+09,9E+09,9E+09,9E+09]];
    CONST robtarget Target_2390:=[[91.252,109.007,3],[0.707106781,0,0,0.707106781],[-1,0,-1,1],[9E+09,9E+09,9E+09,9E+09,9E+09,9E+09]];
    CONST robtarget Target_2400:=[[91.579,110.102,3],[0.707106781,0,0,0.707106781],[-1,0,-1,1],[9E+09,9E+09,9E+09,9E+09,9E+09,9E+09]];
    CONST robtarget Target_2410:=[[91.93,110.81,3],[0.707106781,0,0,0.707106781],[-1,0,-1,1],[9E+09,9E+09,9E+09,9E+09,9E+09,9E+09]];
    CONST robtarget Target_2420:=[[91.895,112.065,3],[0.707106781,0,0,0.707106781],[-1,0,-1,1],[9E+09,9E+09,9E+09,9E+09,9E+09,9E+09]];
    CONST robtarget Target_2430:=[[91.264,113.271,3],[0.707106781,0,0,0.707106781],[-1,0,-1,1],[9E+09,9E+09,9E+09,9E+09,9E+09,9E+09]];
    CONST robtarget Target_2440:=[[90.435,114.264,3],[0.707106781,0,0,0.707106781],[-1,0,-1,1],[9E+09,9E+09,9E+09,9E+09,9E+09,9E+09]];
    CONST robtarget Target_2450:=[[88.968,115.203,3],[0.707106781,0,0,0.707106781],[-1,0,-1,1],[9E+09,9E+09,9E+09,9E+09,9E+09,9E+09]];
    CONST robtarget Target_2460:=[[87.849,115.711,3],[0.707106781,0,0,0.707106781],[-1,0,-1,1],[9E+09,9E+09,9E+09,9E+09,9E+09,9E+09]];
    CONST robtarget Target_2470:=[[86.188,116.255,3],[0.707106781,0,0,0.707106781],[-1,0,-1,1],[9E+09,9E+09,9E+09,9E+09,9E+09,9E+09]];
    CONST robtarget Target_2480:=[[93.07,127.439,-30],[1,0,0,0],[-1,0,-1,1],[9E+09,9E+09,9E+09,9E+09,9E+09,9E+09]];
    CONST robtarget Target_2490:=[[95.469,127.492,0],[1,0,0,0],[-1,0,-1,1],[9E+09,9E+09,9E+09,9E+09,9E+09,9E+09]];
    CONST robtarget Target_2500:=[[141.466,111.749,3],[0.707106781,0,0,0.707106781],[-1,0,-1,1],[9E+09,9E+09,9E+09,9E+09,9E+09,9E+09]];
    CONST robtarget Target_2510:=[[142.181,110.962,3],[0.707106781,0,0,0.707106781],[-1,0,-1,1],[9E+09,9E+09,9E+09,9E+09,9E+09,9E+09]];
    CONST robtarget Target_2520:=[[142.584,110.409,3],[0.707106781,0,0,0.707106781],[-1,0,-1,1],[9E+09,9E+09,9E+09,9E+09,9E+09,9E+09]];
    CONST robtarget Target_2530:=[[143.001,109.909,3],[0.707106781,0,0,0.707106781],[-1,0,-1,1],[9E+09,9E+09,9E+09,9E+09,9E+09,9E+09]];
    CONST robtarget Target_2540:=[[143.755,109.446,3],[0.707106781,0,0,0.707106781],[-1,0,-1,1],[9E+09,9E+09,9E+09,9E+09,9E+09,9E+09]];
    CONST robtarget Target_2550:=[[144.47,108.876,3],[0.707106781,0,0,0.707106781],[-1,0,-1,1],[9E+09,9E+09,9E+09,9E+09,9E+09,9E+09]];
    CONST robtarget Target_2560:=[[144.866,108.509,3],[0.707106781,0,0,0.707106781],[-1,0,-1,1],[9E+09,9E+09,9E+09,9E+09,9E+09,9E+09]];
    CONST robtarget Target_2570:=[[148.292,108.45,3],[0.707106781,0,0,0.707106781],[-1,0,-1,1],[9E+09,9E+09,9E+09,9E+09,9E+09,9E+09]];
    CONST robtarget Target_2580:=[[149.079,109.372,3],[0.707106781,0,0,0.707106781],[-1,0,-1,1],[9E+09,9E+09,9E+09,9E+09,9E+09,9E+09]];
    CONST robtarget Target_2590:=[[149.459,109.996,3],[0.707106781,0,0,0.707106781],[-1,0,-1,1],[9E+09,9E+09,9E+09,9E+09,9E+09,9E+09]];
    CONST robtarget Target_2600:=[[149.804,110.629,3],[0.707106781,0,0,0.707106781],[-1,0,-1,1],[9E+09,9E+09,9E+09,9E+09,9E+09,9E+09]];
    CONST robtarget Target_2610:=[[150.164,111.446,3],[0.707106781,0,0,0.707106781],[-1,0,-1,1],[9E+09,9E+09,9E+09,9E+09,9E+09,9E+09]];
    CONST robtarget Target_2620:=[[150.582,112.397,3],[0.707106781,0,0,0.707106781],[-1,0,-1,1],[9E+09,9E+09,9E+09,9E+09,9E+09,9E+09]];
    CONST robtarget Target_2630:=[[151.11,114.532,3],[0.707106781,0,0,0.707106781],[-1,0,-1,1],[9E+09,9E+09,9E+09,9E+09,9E+09,9E+09]];
    CONST robtarget Target_2640:=[[151.258,118.351,3],[0.707106781,0,0,0.707106781],[-1,0,-1,1],[9E+09,9E+09,9E+09,9E+09,9E+09,9E+09]];
    CONST robtarget Target_2650:=[[151.149,123.493,3],[0.707106781,0,0,0.707106781],[-1,0,-1,1],[9E+09,9E+09,9E+09,9E+09,9E+09,9E+09]];
    CONST robtarget Target_2660:=[[150.509,124.998,3],[0.707106781,0,0,0.707106781],[-1,0,-1,1],[9E+09,9E+09,9E+09,9E+09,9E+09,9E+09]];
    CONST robtarget Target_2670:=[[150.189,126.067,3],[0.707106781,0,0,0.707106781],[-1,0,-1,1],[9E+09,9E+09,9E+09,9E+09,9E+09,9E+09]];
    CONST robtarget Target_2680:=[[119.769,126.854,0],[1,0,0,0],[-1,0,-1,1],[9E+09,9E+09,9E+09,9E+09,9E+09,9E+09]];
    CONST robtarget Target_2690:=[[149.435,127.495,3],[0.707106781,0,0,0.707106781],[-1,0,-1,1],[9E+09,9E+09,9E+09,9E+09,9E+09,9E+09]];
    CONST robtarget Target_2700:=[[149.028,128.307,3],[0.707106781,0,0,0.707106781],[-1,0,-1,1],[9E+09,9E+09,9E+09,9E+09,9E+09,9E+09]];
    CONST robtarget Target_2710:=[[148.353,128.811,3],[0.707106781,0,0,0.707106781],[-1,0,-1,1],[9E+09,9E+09,9E+09,9E+09,9E+09,9E+09]];
    CONST robtarget Target_2720:=[[147.544,129.27,3],[0.707106781,0,0,0.707106781],[-1,0,-1,1],[9E+09,9E+09,9E+09,9E+09,9E+09,9E+09]];
    CONST robtarget Target_2730:=[[146.677,129.693,3],[0.707106781,0,0,0.707106781],[-1,0,-1,1],[9E+09,9E+09,9E+09,9E+09,9E+09,9E+09]];
    CONST robtarget Target_2740:=[[144.048,129.755,3],[0.707106781,0,0,0.707106781],[-1,0,-1,1],[9E+09,9E+09,9E+09,9E+09,9E+09,9E+09]];
    CONST robtarget Target_2750:=[[141.627,127.645,3],[0.707106781,0,0,0.707106781],[-1,0,-1,1],[9E+09,9E+09,9E+09,9E+09,9E+09,9E+09]];
    CONST robtarget Target_2760:=[[171.446,116.13,-27],[0.707106781,0,0,0.707106781],[-1,0,-1,1],[9E+09,9E+09,9E+09,9E+09,9E+09,9E+09]];
    CONST robtarget Target_2770:=[[171.446,116.145,3],[0.707106781,0,0,0.707106781],[-1,0,-1,1],[9E+09,9E+09,9E+09,9E+09,9E+09,9E+09]];
    CONST robtarget Target_2780:=[[171.382,110.454,3],[0.707106781,0,0,0.707106781],[-1,0,-1,1],[9E+09,9E+09,9E+09,9E+09,9E+09,9E+09]];
    CONST robtarget Target_2790:=[[172.421,109.424,3],[0.707106781,0,0,0.707106781],[-1,0,-1,1],[9E+09,9E+09,9E+09,9E+09,9E+09,9E+09]];
    CONST robtarget Target_2800:=[[173.527,108.448,3],[0.707106781,0,0,0.707106781],[-1,0,-1,1],[9E+09,9E+09,9E+09,9E+09,9E+09,9E+09]];
    CONST robtarget Target_2810:=[[174.583,107.985,3],[0.707106781,0,0,0.707106781],[-1,0,-1,1],[9E+09,9E+09,9E+09,9E+09,9E+09,9E+09]];
    CONST robtarget Target_2820:=[[175.225,107.505,3],[0.707106781,0,0,0.707106781],[-1,0,-1,1],[9E+09,9E+09,9E+09,9E+09,9E+09,9E+09]];
    CONST robtarget Target_2830:=[[178.189,107.549,3],[0.707106781,0,0,0.707106781],[-1,0,-1,1],[9E+09,9E+09,9E+09,9E+09,9E+09,9E+09]];
    CONST robtarget Target_2840:=[[178.951,108.484,3],[0.707106781,0,0,0.707106781],[-1,0,-1,1],[9E+09,9E+09,9E+09,9E+09,9E+09,9E+09]];
    CONST robtarget Target_2850:=[[179.322,108.956,3],[0.707106781,0,0,0.707106781],[-1,0,-1,1],[9E+09,9E+09,9E+09,9E+09,9E+09,9E+09]];
    CONST robtarget Target_2860:=[[179.662,109.677,3],[0.707106781,0,0,0.707106781],[-1,0,-1,1],[9E+09,9E+09,9E+09,9E+09,9E+09,9E+09]];
    CONST robtarget Target_2870:=[[179.673,112.896,3],[0.707106781,0,0,0.707106781],[-1,0,-1,1],[9E+09,9E+09,9E+09,9E+09,9E+09,9E+09]];
    CONST robtarget Target_2880:=[[178.94,113.73,3],[0.707106781,0,0,0.707106781],[-1,0,-1,1],[9E+09,9E+09,9E+09,9E+09,9E+09,9E+09]];
    CONST robtarget Target_2890:=[[177.839,114.708,3],[0.707106781,0,0,0.707106781],[-1,0,-1,1],[9E+09,9E+09,9E+09,9E+09,9E+09,9E+09]];
    CONST robtarget Target_2900:=[[175.361,115.711,3],[0.707106781,0,0,0.707106781],[-1,0,-1,1],[9E+09,9E+09,9E+09,9E+09,9E+09,9E+09]];
    CONST robtarget Target_2910:=[[174.498,116.176,3],[0.707106781,0,0,0.707106781],[-1,0,-1,1],[9E+09,9E+09,9E+09,9E+09,9E+09,9E+09]];
    PERS tooldata Soporte_final:=[TRUE,[[114.807,-0.025,36.238],[0.5,0,0.866025,0]],[1,[0,0,1],[1,0,0,0],0,0,0]];
    TASK PERS wobjdata ADwob:=[FALSE,TRUE,"",[[-100,-130,-20],[1,0,0,0]],[[280,-670,540],[0,0,1,0]]];
    CONST robtarget Target_minihome_2:=[[140,90,-100],[0.707106781,0,0,0.707106781],[-1,0,-1,1],[9E+09,9E+09,9E+09,9E+09,9E+09,9E+09]];
    CONST robtarget Target_3020:=[[40.936,101.854,0],[0.707106781,0,0,0.707106781],[-1,0,-1,1],[9E+09,9E+09,9E+09,9E+09,9E+09,9E+09]];
    CONST robtarget Target_2920_up:=[[207.225,82.129060431,-27.180922138],[0.69636424,-0.122787804,0.122787804,0.69636424],[-2,-1,0,1],[9E+09,9E+09,9E+09,9E+09,9E+09,9E+09]];
    CONST robtarget Target_2920:=[[207.225,82.129060431,2.819077862],[0.69636424,-0.122787804,0.122787804,0.69636424],[-2,-1,0,1],[9E+09,9E+09,9E+09,9E+09,9E+09,9E+09]];
    CONST robtarget Target_2930:=[[189.302,82.034060431,2.819077862],[0.69636424,-0.122787804,0.122787804,0.69636424],[-2,-1,0,1],[9E+09,9E+09,9E+09,9E+09,9E+09,9E+09]];
    CONST robtarget Target_2940:=[[172.295,56.628060431,2.819077862],[0.69636424,-0.122787804,0.122787804,0.69636424],[-1,0,-1,1],[9E+09,9E+09,9E+09,9E+09,9E+09,9E+09]];
    CONST robtarget Target_2950:=[[189.448,31.520060431,2.819077862],[0.69636424,-0.122787804,0.122787804,0.69636424],[-2,-1,0,1],[9E+09,9E+09,9E+09,9E+09,9E+09,9E+09]];
    CONST robtarget Target_2960:=[[207.063,31.366060431,2.819077862],[0.69636424,-0.122787804,0.122787804,0.69636424],[-2,-1,0,1],[9E+09,9E+09,9E+09,9E+09,9E+09,9E+09]];
    CONST robtarget Target_2970_up:=[[198.201,73.121060431,-27.180922138],[0.69636424,-0.122787804,0.122787804,0.69636424],[-2,-1,0,1],[9E+09,9E+09,9E+09,9E+09,9E+09,9E+09]];
    CONST robtarget Target_2970:=[[198.201,73.121060431,2.819077862],[0.69636424,-0.122787804,0.122787804,0.69636424],[-2,-1,0,1],[9E+09,9E+09,9E+09,9E+09,9E+09,9E+09]];
    CONST robtarget Target_2980:=[[189.482,72.946060431,2.819077862],[0.69636424,-0.122787804,0.122787804,0.69636424],[-2,-1,0,1],[9E+09,9E+09,9E+09,9E+09,9E+09,9E+09]];
    CONST robtarget Target_2990:=[[181.283,56.738060431,2.819077862],[0.69636424,-0.122787804,0.122787804,0.69636424],[-2,-1,0,1],[9E+09,9E+09,9E+09,9E+09,9E+09,9E+09]];
    CONST robtarget Target_3000:=[[189.826,40.515060431,2.819077862],[0.69636424,-0.122787804,0.122787804,0.69636424],[-2,-1,0,1],[9E+09,9E+09,9E+09,9E+09,9E+09,9E+09]];
    CONST robtarget Target_3010:=[[198.134,40.185060431,2.819077862],[0.69636424,-0.122787804,0.122787804,0.69636424],[-2,-1,0,1],[9E+09,9E+09,9E+09,9E+09,9E+09,9E+09]];
    CONST robtarget Target_3030_2:=[[168.856,62.045020144,-29.060307379],[0.69636424,-0.122787804,0.122787804,0.69636424],[-1,0,-1,1],[9E+09,9E+09,9E+09,9E+09,9E+09,9E+09]];
    CONST robtarget Target_3030:=[[168.856,62.729060431,2.819077862],[0.69636424,-0.122787804,0.122787804,0.69636424],[-1,0,-1,1],[9E+09,9E+09,9E+09,9E+09,9E+09,9E+09]];
    CONST robtarget Target_3040:=[[164.492,65.336020144,0.939692621],[0.69636424,-0.122787804,0.122787804,0.69636424],[-1,0,-1,1],[9E+09,9E+09,9E+09,9E+09,9E+09,9E+09]];
    CONST robtarget Target_3050:=[[159.783,67.041020144,0.939692621],[0.69636424,-0.122787804,0.122787804,0.69636424],[-1,0,-1,1],[9E+09,9E+09,9E+09,9E+09,9E+09,9E+09]];
    CONST robtarget Target_3060:=[[154.529,67.248020144,0.939692621],[0.69636424,-0.122787804,0.122787804,0.69636424],[-1,0,-1,1],[9E+09,9E+09,9E+09,9E+09,9E+09,9E+09]];
    CONST robtarget Target_3070:=[[149.168,63.265020144,0.939692621],[0.69636424,-0.122787804,0.122787804,0.69636424],[-1,0,-1,1],[9E+09,9E+09,9E+09,9E+09,9E+09,9E+09]];
    CONST robtarget Target_3080:=[[146.594,56.470020144,0.939692621],[0.69636424,-0.122787804,0.122787804,0.69636424],[-1,0,-1,1],[9E+09,9E+09,9E+09,9E+09,9E+09,9E+09]];
    CONST robtarget Target_3090:=[[146.435,30.622020144,0.939692621],[0.69636424,-0.122787804,0.122787804,0.69636424],[-1,0,-1,1],[9E+09,9E+09,9E+09,9E+09,9E+09,9E+09]];
    CONST robtarget Target_3100:=[[151.326,30.602020144,0.939692621],[0.69636424,-0.122787804,0.122787804,0.69636424],[-1,0,-1,1],[9E+09,9E+09,9E+09,9E+09,9E+09,9E+09]];
    CONST robtarget Target_3110:=[[153.44,34.909020144,0.939692621],[0.69636424,-0.122787804,0.122787804,0.69636424],[-1,0,-1,1],[9E+09,9E+09,9E+09,9E+09,9E+09,9E+09]];
    CONST robtarget Target_3120:=[[156.57,31.843020144,0.939692621],[0.69636424,-0.122787804,0.122787804,0.69636424],[-1,0,-1,1],[9E+09,9E+09,9E+09,9E+09,9E+09,9E+09]];
    CONST robtarget Target_3130:=[[160.302,30.191020144,0.939692621],[0.69636424,-0.122787804,0.122787804,0.69636424],[-1,0,-1,1],[9E+09,9E+09,9E+09,9E+09,9E+09,9E+09]];
    CONST robtarget Target_3140:=[[163.825,30.168020144,0.939692621],[0.69636424,-0.122787804,0.122787804,0.69636424],[-1,0,-1,1],[9E+09,9E+09,9E+09,9E+09,9E+09,9E+09]];
    CONST robtarget Target_3150:=[[167.12,31.969020144,0.939692621],[0.69636424,-0.122787804,0.122787804,0.69636424],[-1,0,-1,1],[9E+09,9E+09,9E+09,9E+09,9E+09,9E+09]];
    CONST robtarget Target_3160:=[[169.87,36.987020144,0.939692621],[0.69636424,-0.122787804,0.122787804,0.69636424],[-1,0,-1,1],[9E+09,9E+09,9E+09,9E+09,9E+09,9E+09]];
    CONST robtarget Target_3170:=[[170.005,41.186020144,0.939692621],[0.69636424,-0.122787804,0.122787804,0.69636424],[-1,0,-1,1],[9E+09,9E+09,9E+09,9E+09,9E+09,9E+09]];
    CONST robtarget Target_3180:=[[166.518,48.057020144,0.939692621],[0.69636424,-0.122787804,0.122787804,0.69636424],[-1,0,-1,1],[9E+09,9E+09,9E+09,9E+09,9E+09,9E+09]];
    CONST robtarget Target_3190:=[[159.562,51.317020144,0.939692621],[0.69636424,-0.122787804,0.122787804,0.69636424],[-1,0,-1,1],[9E+09,9E+09,9E+09,9E+09,9E+09,9E+09]];
    CONST robtarget Target_3200:=[[154.356,51.836020144,0.939692621],[0.69636424,-0.122787804,0.122787804,0.69636424],[-1,0,-1,1],[9E+09,9E+09,9E+09,9E+09,9E+09,9E+09]];
    CONST robtarget Target_3210:=[[154.402,56.254020144,0.939692621],[0.69636424,-0.122787804,0.122787804,0.69636424],[-1,0,-1,1],[9E+09,9E+09,9E+09,9E+09,9E+09,9E+09]];
    CONST robtarget Target_3220:=[[156.646,59.021020144,0.939692621],[0.69636424,-0.122787804,0.122787804,0.69636424],[-1,0,-1,1],[9E+09,9E+09,9E+09,9E+09,9E+09,9E+09]];
    CONST robtarget Target_3230:=[[159.999,59.059020144,0.939692621],[0.69636424,-0.122787804,0.122787804,0.69636424],[-1,0,-1,1],[9E+09,9E+09,9E+09,9E+09,9E+09,9E+09]];
    CONST robtarget Target_3240:=[[163.724,56.946020144,0.939692621],[0.69636424,-0.122787804,0.122787804,0.69636424],[-1,0,-1,1],[9E+09,9E+09,9E+09,9E+09,9E+09,9E+09]];
    CONST robtarget Target_3250:=[[166.309,56.964020144,0.939692621],[0.69636424,-0.122787804,0.122787804,0.69636424],[-1,0,-1,1],[9E+09,9E+09,9E+09,9E+09,9E+09,9E+09]];
    CONST robtarget Target_3260_2:=[[154.254,45.587020144,-29.060307379],[0.69636424,-0.122787804,0.122787804,0.69636424],[-1,0,-1,1],[9E+09,9E+09,9E+09,9E+09,9E+09,9E+09]];
    CONST robtarget Target_3260:=[[154.254,45.587020144,0.939692621],[0.69636424,-0.122787804,0.122787804,0.69636424],[-1,0,-1,1],[9E+09,9E+09,9E+09,9E+09,9E+09,9E+09]];
    CONST robtarget Target_3270:=[[154.243,40.170020144,0.939692621],[0.69636424,-0.122787804,0.122787804,0.69636424],[-1,0,-1,1],[9E+09,9E+09,9E+09,9E+09,9E+09,9E+09]];
    CONST robtarget Target_3280:=[[155.887,38.274020144,0.939692621],[0.69636424,-0.122787804,0.122787804,0.69636424],[-1,0,-1,1],[9E+09,9E+09,9E+09,9E+09,9E+09,9E+09]];
    CONST robtarget Target_3290:=[[157.675,37.336020144,0.939692621],[0.69636424,-0.122787804,0.122787804,0.69636424],[-1,0,-1,1],[9E+09,9E+09,9E+09,9E+09,9E+09,9E+09]];
    CONST robtarget Target_3300:=[[160.603,37.207020144,0.939692621],[0.69636424,-0.122787804,0.122787804,0.69636424],[-1,0,-1,1],[9E+09,9E+09,9E+09,9E+09,9E+09,9E+09]];
    CONST robtarget Target_3310:=[[162.533,39.193020144,0.939692621],[0.69636424,-0.122787804,0.122787804,0.69636424],[-1,0,-1,1],[9E+09,9E+09,9E+09,9E+09,9E+09,9E+09]];
    CONST robtarget Target_3320:=[[162.426,41.941020144,0.939692621],[0.69636424,-0.122787804,0.122787804,0.69636424],[-1,0,-1,1],[9E+09,9E+09,9E+09,9E+09,9E+09,9E+09]];
    CONST robtarget Target_3330:=[[160.229,44.430020144,0.939692621],[0.69636424,-0.122787804,0.122787804,0.69636424],[-1,0,-1,1],[9E+09,9E+09,9E+09,9E+09,9E+09,9E+09]];
    CONST robtarget Target_3340:=[[157.734,45.576020144,0.939692621],[0.69636424,-0.122787804,0.122787804,0.69636424],[-1,0,-1,1],[9E+09,9E+09,9E+09,9E+09,9E+09,9E+09]];
    CONST robtarget Target_3350_2:=[[144.461,67.032020144,-29.060307379],[0.69636424,-0.122787804,0.122787804,0.69636424],[-1,0,-1,1],[9E+09,9E+09,9E+09,9E+09,9E+09,9E+09]];
    CONST robtarget Target_3350:=[[144.461,67.032020144,0.939692621],[0.69636424,-0.122787804,0.122787804,0.69636424],[-1,0,-1,1],[9E+09,9E+09,9E+09,9E+09,9E+09,9E+09]];
    CONST robtarget Target_3360:=[[136.399,66.775020144,0.939692621],[0.69636424,-0.122787804,0.122787804,0.69636424],[-1,0,-1,1],[9E+09,9E+09,9E+09,9E+09,9E+09,9E+09]];
    CONST robtarget Target_3370:=[[130.223,41.577020144,0.939692621],[0.69636424,-0.122787804,0.122787804,0.69636424],[-1,0,-1,1],[9E+09,9E+09,9E+09,9E+09,9E+09,9E+09]];
    CONST robtarget Target_3380:=[[123.937,66.551020144,0.939692621],[0.69636424,-0.122787804,0.122787804,0.69636424],[-1,0,-1,1],[9E+09,9E+09,9E+09,9E+09,9E+09,9E+09]];
    CONST robtarget Target_3390:=[[115.96,66.627020144,0.939692621],[0.69636424,-0.122787804,0.122787804,0.69636424],[-1,0,-1,1],[9E+09,9E+09,9E+09,9E+09,9E+09,9E+09]];
    CONST robtarget Target_3400:=[[126.475,30.638020144,0.939692621],[0.69636424,-0.122787804,0.122787804,0.69636424],[-1,0,-1,1],[9E+09,9E+09,9E+09,9E+09,9E+09,9E+09]];
    CONST robtarget Target_3410:=[[133.864,30.673020144,0.939692621],[0.69636424,-0.122787804,0.122787804,0.69636424],[-1,0,-1,1],[9E+09,9E+09,9E+09,9E+09,9E+09,9E+09]];
    CONST robtarget Target_3420_2:=[[112.825,66.820020144,-29.060307379],[0.69636424,-0.122787804,0.122787804,0.69636424],[-1,0,-1,1],[9E+09,9E+09,9E+09,9E+09,9E+09,9E+09]];
    CONST robtarget Target_3420:=[[112.825,66.820020144,0.939692621],[0.69636424,-0.122787804,0.122787804,0.69636424],[-1,0,-1,1],[9E+09,9E+09,9E+09,9E+09,9E+09,9E+09]];
    CONST robtarget Target_3430:=[[104.746,66.822020144,0.939692621],[0.69636424,-0.122787804,0.122787804,0.69636424],[-1,0,-1,1],[9E+09,9E+09,9E+09,9E+09,9E+09,9E+09]];
    CONST robtarget Target_3440:=[[104.632,30.482020144,0.939692621],[0.69636424,-0.122787804,0.122787804,0.69636424],[-1,0,-1,1],[9E+09,9E+09,9E+09,9E+09,9E+09,9E+09]];
    CONST robtarget Target_3450:=[[112.782,30.740020144,0.939692621],[0.69636424,-0.122787804,0.122787804,0.69636424],[-1,0,-1,1],[9E+09,9E+09,9E+09,9E+09,9E+09,9E+09]];
    CONST robtarget Target_3460_2:=[[107.732,82.799020144,-29.060307379],[0.69636424,-0.122787804,0.122787804,0.69636424],[-1,0,-1,1],[9E+09,9E+09,9E+09,9E+09,9E+09,9E+09]];
    CONST robtarget Target_3460:=[[107.732,82.799020144,0.939692621],[0.69636424,-0.122787804,0.122787804,0.69636424],[-1,0,-1,1],[9E+09,9E+09,9E+09,9E+09,9E+09,9E+09]];
    CONST robtarget Target_3470:=[[103.914,76.496020144,0.939692621],[0.69636424,-0.122787804,0.122787804,0.69636424],[-1,0,-1,1],[9E+09,9E+09,9E+09,9E+09,9E+09,9E+09]];
    CONST robtarget Target_3480:=[[107.812,70.304020144,0.939692621],[0.69636424,-0.122787804,0.122787804,0.69636424],[-1,0,-1,1],[9E+09,9E+09,9E+09,9E+09,9E+09,9E+09]];
    CONST robtarget Target_3490:=[[110.105,70.397020144,0.939692621],[0.69636424,-0.122787804,0.122787804,0.69636424],[-1,0,-1,1],[9E+09,9E+09,9E+09,9E+09,9E+09,9E+09]];
    CONST robtarget Target_3500:=[[113.61,76.180020144,0.939692621],[0.69636424,-0.122787804,0.122787804,0.69636424],[-1,0,-1,1],[9E+09,9E+09,9E+09,9E+09,9E+09,9E+09]];
    CONST robtarget Target_3510:=[[110.04,82.825020144,0.939692621],[0.69636424,-0.122787804,0.122787804,0.69636424],[-1,0,-1,1],[9E+09,9E+09,9E+09,9E+09,9E+09,9E+09]];
    CONST robtarget Target_3520_2:=[[82.277,82.761020144,-29.060307379],[0.69636424,-0.122787804,0.122787804,0.69636424],[-1,0,-1,1],[9E+09,9E+09,9E+09,9E+09,9E+09,9E+09]];
    CONST robtarget Target_3520:=[[82.277,82.761020144,0.939692621],[0.69636424,-0.122787804,0.122787804,0.69636424],[-1,0,-1,1],[9E+09,9E+09,9E+09,9E+09,9E+09,9E+09]];
    CONST robtarget Target_3530:=[[74.455,82.673020144,0.939692621],[0.69636424,-0.122787804,0.122787804,0.69636424],[-1,0,-1,1],[9E+09,9E+09,9E+09,9E+09,9E+09,9E+09]];
    CONST robtarget Target_3540:=[[74.428,30.709020144,0.939692621],[0.69636424,-0.122787804,0.122787804,0.69636424],[-1,0,-1,1],[9E+09,9E+09,9E+09,9E+09,9E+09,9E+09]];
    CONST robtarget Target_3550:=[[80.004,30.702020144,0.939692621],[0.69636424,-0.122787804,0.122787804,0.69636424],[-1,0,-1,1],[9E+09,9E+09,9E+09,9E+09,9E+09,9E+09]];
    CONST robtarget Target_3560:=[[82.07,35.013020144,0.939692621],[0.69636424,-0.122787804,0.122787804,0.69636424],[-1,0,-1,1],[9E+09,9E+09,9E+09,9E+09,9E+09,9E+09]];
    CONST robtarget Target_3570:=[[84.954,31.898020144,0.939692621],[0.69636424,-0.122787804,0.122787804,0.69636424],[-1,0,-1,1],[9E+09,9E+09,9E+09,9E+09,9E+09,9E+09]];
    CONST robtarget Target_3580:=[[88.431,30.331020144,0.939692621],[0.69636424,-0.122787804,0.122787804,0.69636424],[-1,0,-1,1],[9E+09,9E+09,9E+09,9E+09,9E+09,9E+09]];
    CONST robtarget Target_3590:=[[92.072,30.216020144,0.939692621],[0.69636424,-0.122787804,0.122787804,0.69636424],[-1,0,-1,1],[9E+09,9E+09,9E+09,9E+09,9E+09,9E+09]];
    CONST robtarget Target_3600:=[[97.435,34.873020144,0.939692621],[0.69636424,-0.122787804,0.122787804,0.69636424],[-1,0,-1,1],[9E+09,9E+09,9E+09,9E+09,9E+09,9E+09]];
    CONST robtarget Target_3610:=[[99.865,42.963020144,0.939692621],[0.69636424,-0.122787804,0.122787804,0.69636424],[-1,0,-1,1],[9E+09,9E+09,9E+09,9E+09,9E+09,9E+09]];
    CONST robtarget Target_3620:=[[100.165,49.389020144,0.939692621],[0.69636424,-0.122787804,0.122787804,0.69636424],[-1,0,-1,1],[9E+09,9E+09,9E+09,9E+09,9E+09,9E+09]];
    CONST robtarget Target_3630:=[[97.664,60.583020144,0.939692621],[0.69636424,-0.122787804,0.122787804,0.69636424],[-1,0,-1,1],[9E+09,9E+09,9E+09,9E+09,9E+09,9E+09]];
    CONST robtarget Target_3640:=[[90.704,67.178020144,0.939692621],[0.69636424,-0.122787804,0.122787804,0.69636424],[-1,0,-1,1],[9E+09,9E+09,9E+09,9E+09,9E+09,9E+09]];
    CONST robtarget Target_3650:=[[86.592,67.289020144,0.939692621],[0.69636424,-0.122787804,0.122787804,0.69636424],[-1,0,-1,1],[9E+09,9E+09,9E+09,9E+09,9E+09,9E+09]];
    CONST robtarget Target_3660:=[[82.282,64.136020144,0.939692621],[0.69636424,-0.122787804,0.122787804,0.69636424],[-1,0,-1,1],[9E+09,9E+09,9E+09,9E+09,9E+09,9E+09]];
    CONST robtarget Target_3670_2:=[[82.253,56.509020144,-29.060307379],[0.69636424,-0.122787804,0.122787804,0.69636424],[-1,0,-1,1],[9E+09,9E+09,9E+09,9E+09,9E+09,9E+09]];
    CONST robtarget Target_3670:=[[82.253,56.509020144,0.939692621],[0.69636424,-0.122787804,0.122787804,0.69636424],[-1,0,-1,1],[9E+09,9E+09,9E+09,9E+09,9E+09,9E+09]];
    CONST robtarget Target_3680:=[[82.272,41.520020144,0.939692621],[0.69636424,-0.122787804,0.122787804,0.69636424],[-1,0,-1,1],[9E+09,9E+09,9E+09,9E+09,9E+09,9E+09]];
    CONST robtarget Target_3690:=[[85.391,38.217020144,0.939692621],[0.69636424,-0.122787804,0.122787804,0.69636424],[-1,0,-1,1],[9E+09,9E+09,9E+09,9E+09,9E+09,9E+09]];
    CONST robtarget Target_3700:=[[88.811,38.071020144,0.939692621],[0.69636424,-0.122787804,0.122787804,0.69636424],[-1,0,-1,1],[9E+09,9E+09,9E+09,9E+09,9E+09,9E+09]];
    CONST robtarget Target_3710:=[[91.889,43.979020144,0.939692621],[0.69636424,-0.122787804,0.122787804,0.69636424],[-1,0,-1,1],[9E+09,9E+09,9E+09,9E+09,9E+09,9E+09]];
    CONST robtarget Target_3720:=[[92.083,51.104020144,0.939692621],[0.69636424,-0.122787804,0.122787804,0.69636424],[-1,0,-1,1],[9E+09,9E+09,9E+09,9E+09,9E+09,9E+09]];
    CONST robtarget Target_3730:=[[89.43,58.065020144,0.939692621],[0.69636424,-0.122787804,0.122787804,0.69636424],[-1,0,-1,1],[9E+09,9E+09,9E+09,9E+09,9E+09,9E+09]];
    CONST robtarget Target_3740:=[[85.526,58.965020144,0.939692621],[0.69636424,-0.122787804,0.122787804,0.69636424],[-1,0,-1,1],[9E+09,9E+09,9E+09,9E+09,9E+09,9E+09]];
    CONST robtarget Target_3750:=[[64.524,146.437020144,0.939692621],[0.69636424,-0.122787804,0.122787804,0.69636424],[-1,0,-1,1],[9E+09,9E+09,9E+09,9E+09,9E+09,9E+09]];
    CONST robtarget Target_3750_2:=[[64.524,146.437020144,-29.060307379],[0.69636424,-0.122787804,0.122787804,0.69636424],[-1,0,-1,1],[9E+09,9E+09,9E+09,9E+09,9E+09,9E+09]];
    CONST robtarget Target_3760:=[[55.549,133.666020144,0.939692621],[0.69636424,-0.122787804,0.122787804,0.69636424],[-1,0,-1,1],[9E+09,9E+09,9E+09,9E+09,9E+09,9E+09]];
    CONST robtarget Target_3770:=[[47.044,128.487020144,0.939692621],[0.69636424,-0.122787804,0.122787804,0.69636424],[-1,0,-1,1],[9E+09,9E+09,9E+09,9E+09,9E+09,9E+09]];
    CONST robtarget Target_3780:=[[37.688,111.228020144,0.939692621],[0.69636424,-0.122787804,0.122787804,0.69636424],[-1,0,-1,1],[9E+09,9E+09,9E+09,9E+09,9E+09,9E+09]];
    CONST robtarget Target_3790:=[[41.259,123.994020144,0.939692621],[0.69636424,-0.122787804,0.122787804,0.69636424],[-1,0,-1,1],[9E+09,9E+09,9E+09,9E+09,9E+09,9E+09]];
    CONST robtarget Target_3800:=[[26.923,126.980020144,0.939692621],[0.69636424,-0.122787804,0.122787804,0.69636424],[-1,0,-1,1],[9E+09,9E+09,9E+09,9E+09,9E+09,9E+09]];
    CONST robtarget Target_3810:=[[26.91,85.429020144,0.939692621],[0.69636424,-0.122787804,0.122787804,0.69636424],[-1,0,-1,1],[9E+09,9E+09,9E+09,9E+09,9E+09,9E+09]];
    CONST robtarget Target_3820:=[[31.003,81.597020144,0.939692621],[0.69636424,-0.122787804,0.122787804,0.69636424],[-1,0,-1,1],[9E+09,9E+09,9E+09,9E+09,9E+09,9E+09]];
    CONST robtarget Target_3830:=[[35.653,89.236020144,0.939692621],[0.69636424,-0.122787804,0.122787804,0.69636424],[-1,0,-1,1],[9E+09,9E+09,9E+09,9E+09,9E+09,9E+09]];
    CONST robtarget Target_3840:=[[41.161,97.045020144,0.939692621],[0.69636424,-0.122787804,0.122787804,0.69636424],[-1,0,-1,1],[9E+09,9E+09,9E+09,9E+09,9E+09,9E+09]];
    CONST robtarget Target_3850:=[[45.695,102.026020144,0.939692621],[0.69636424,-0.122787804,0.122787804,0.69636424],[-1,0,-1,1],[9E+09,9E+09,9E+09,9E+09,9E+09,9E+09]];
    CONST robtarget Target_3860:=[[52.946,106.880020144,0.939692621],[0.69636424,-0.122787804,0.122787804,0.69636424],[-1,0,-1,1],[9E+09,9E+09,9E+09,9E+09,9E+09,9E+09]];
    CONST robtarget Target_3870:=[[62.408,123.824020144,0.939692621],[0.69636424,-0.122787804,0.122787804,0.69636424],[-1,0,-1,1],[9E+09,9E+09,9E+09,9E+09,9E+09,9E+09]];
    CONST robtarget Target_3880:=[[52.276,112.163020144,0.939692621],[0.69636424,-0.122787804,0.122787804,0.69636424],[-1,0,-1,1],[9E+09,9E+09,9E+09,9E+09,9E+09,9E+09]];
    CONST robtarget Target_3890:=[[59.313,122.581020144,0.939692621],[0.69636424,-0.122787804,0.122787804,0.69636424],[-1,0,-1,1],[9E+09,9E+09,9E+09,9E+09,9E+09,9E+09]];
    CONST robtarget Target_3900:=[[63.763,135.404020144,0.939692621],[0.69636424,-0.122787804,0.122787804,0.69636424],[-1,0,-1,1],[9E+09,9E+09,9E+09,9E+09,9E+09,9E+09]];
    CONST robtarget Target_3910:=[[27.611,83.068020144,0.939692621],[0.69636424,-0.122787804,0.122787804,0.69636424],[-1,0,-1,1],[9E+09,9E+09,9E+09,9E+09,9E+09,9E+09]];
    CONST robtarget Target_3910_2:=[[27.611,83.068020144,-29.060307379],[0.69636424,-0.122787804,0.122787804,0.69636424],[-1,0,-1,1],[9E+09,9E+09,9E+09,9E+09,9E+09,9E+09]];
    CONST robtarget Target_3920:=[[24.514,80.149020144,0.939692621],[0.69636424,-0.122787804,0.122787804,0.69636424],[-1,0,-1,1],[9E+09,9E+09,9E+09,9E+09,9E+09,9E+09]];
    CONST robtarget Target_3930:=[[24.493,70.759020144,0.939692621],[0.69636424,-0.122787804,0.122787804,0.69636424],[-1,0,-1,1],[9E+09,9E+09,9E+09,9E+09,9E+09,9E+09]];
    CONST robtarget Target_3940:=[[26.846,61.477020144,0.939692621],[0.69636424,-0.122787804,0.122787804,0.69636424],[-1,0,-1,1],[9E+09,9E+09,9E+09,9E+09,9E+09,9E+09]];
    CONST robtarget Target_3950:=[[29.828,69.272020144,0.939692621],[0.69636424,-0.122787804,0.122787804,0.69636424],[-1,0,-1,1],[9E+09,9E+09,9E+09,9E+09,9E+09,9E+09]];
    CONST robtarget Target_3960:=[[30.012,78.359020144,0.939692621],[0.69636424,-0.122787804,0.122787804,0.69636424],[-1,0,-1,1],[9E+09,9E+09,9E+09,9E+09,9E+09,9E+09]];
    CONST robtarget Target_3970:=[[44.273,96.711020144,0.939692621],[0.69636424,-0.122787804,0.122787804,0.69636424],[-1,0,-1,1],[9E+09,9E+09,9E+09,9E+09,9E+09,9E+09]];
    CONST robtarget Target_3970_2:=[[44.273,96.711020144,-29.060307379],[0.69636424,-0.122787804,0.122787804,0.69636424],[-1,0,-1,1],[9E+09,9E+09,9E+09,9E+09,9E+09,9E+09]];
    CONST robtarget Target_3980:=[[43.933,86.227020144,0.939692621],[0.69636424,-0.122787804,0.122787804,0.69636424],[-1,0,-1,1],[9E+09,9E+09,9E+09,9E+09,9E+09,9E+09]];
    CONST robtarget Target_3990:=[[39.768,82.418020144,0.939692621],[0.69636424,-0.122787804,0.122787804,0.69636424],[-1,0,-1,1],[9E+09,9E+09,9E+09,9E+09,9E+09,9E+09]];
    CONST robtarget Target_4000:=[[34.596,82.452020144,0.939692621],[0.69636424,-0.122787804,0.122787804,0.69636424],[-1,0,-1,1],[9E+09,9E+09,9E+09,9E+09,9E+09,9E+09]];
    CONST robtarget Target_4010:=[[26.792,57.803020144,0.939692621],[0.69636424,-0.122787804,0.122787804,0.69636424],[-1,0,-1,1],[9E+09,9E+09,9E+09,9E+09,9E+09,9E+09]];
    CONST robtarget Target_4010_2:=[[26.792,57.803020144,-29.060307379],[0.69636424,-0.122787804,0.122787804,0.69636424],[-1,0,-1,1],[9E+09,9E+09,9E+09,9E+09,9E+09,9E+09]];
    CONST robtarget Target_4020:=[[45.072,60.926020144,0.939692621],[0.69636424,-0.122787804,0.122787804,0.69636424],[-1,0,-1,1],[9E+09,9E+09,9E+09,9E+09,9E+09,9E+09]];
    CONST robtarget Target_4030:=[[61.878,52.724020144,0.939692621],[0.69636424,-0.122787804,0.122787804,0.69636424],[-1,0,-1,1],[9E+09,9E+09,9E+09,9E+09,9E+09,9E+09]];
    CONST robtarget Target_4040:=[[59.898,63.620020144,0.939692621],[0.69636424,-0.122787804,0.122787804,0.69636424],[-1,0,-1,1],[9E+09,9E+09,9E+09,9E+09,9E+09,9E+09]];
    CONST robtarget Target_4050:=[[56.445,72.459020144,0.939692621],[0.69636424,-0.122787804,0.122787804,0.69636424],[-1,0,-1,1],[9E+09,9E+09,9E+09,9E+09,9E+09,9E+09]];
    CONST robtarget Target_4060:=[[58.835,86.000020144,0.939692621],[0.69636424,-0.122787804,0.122787804,0.69636424],[-1,0,-1,1],[9E+09,9E+09,9E+09,9E+09,9E+09,9E+09]];
    CONST robtarget Target_4070:=[[54.916,107.364020144,0.939692621],[0.69636424,-0.122787804,0.122787804,0.69636424],[-1,0,-1,1],[9E+09,9E+09,9E+09,9E+09,9E+09,9E+09]];
    CONST robtarget Target_4080:=[[49.508,100.246020144,0.939692621],[0.69636424,-0.122787804,0.122787804,0.69636424],[-1,0,-1,1],[9E+09,9E+09,9E+09,9E+09,9E+09,9E+09]];
    CONST robtarget Target_4090:=[[52.038,93.753020144,0.939692621],[0.69636424,-0.122787804,0.122787804,0.69636424],[-1,0,-1,1],[9E+09,9E+09,9E+09,9E+09,9E+09,9E+09]];
    CONST robtarget Target_4100:=[[52.392,84.414020144,0.939692621],[0.69636424,-0.122787804,0.122787804,0.69636424],[-1,0,-1,1],[9E+09,9E+09,9E+09,9E+09,9E+09,9E+09]];
    CONST robtarget Target_4110:=[[48.592,78.019020144,0.939692621],[0.69636424,-0.122787804,0.122787804,0.69636424],[-1,0,-1,1],[9E+09,9E+09,9E+09,9E+09,9E+09,9E+09]];
    CONST robtarget Target_4120:=[[44.019,73.976020144,0.939692621],[0.69636424,-0.122787804,0.122787804,0.69636424],[-1,0,-1,1],[9E+09,9E+09,9E+09,9E+09,9E+09,9E+09]];
    CONST robtarget Target_4130:=[[36.693,67.321020144,0.939692621],[0.69636424,-0.122787804,0.122787804,0.69636424],[-1,0,-1,1],[9E+09,9E+09,9E+09,9E+09,9E+09,9E+09]];
    CONST robtarget Target_Home:=[[-200.271,669.975,-21.956],[0.866025404,0,0.5,0],[0,0,0,0],[9E+09,9E+09,9E+09,9E+09,9E+09,9E+09]];
    CONST jointtarget HOME_Origen:=[[0,0,0,0,0,0],[9E+09,9E+09,9E+09,9E+09,9E+09,9E+09]];
    CONST jointtarget RomperSingular:=[[0,0,0,0,30,0],[9E+09,9E+09,9E+09,9E+09,9E+09,9E+09]];
    CONST jointtarget cambio_Tool:=[[80,0,0,0,-45,45],[9E+09,9E+09,9E+09,9E+09,9E+09,9E+09]];



    PROC main()
        TPErase;
        TPWrite "Iniciando Ciclo";
        !Aquí se reinicia todas las entradas y salidad a usar.
        Reset Conveyor_FWD;
        Reset Conveyor_INV;
        Reset DO_01;
        Reset DO_02;
        GoHome;
        TPWrite "Porfavor presione Botón1 para iniciar Rutina de decoración ";
        TPWrite "Tambien, puede presionar Botón2 para iniciar Rutina de Matenimiento ";

   WHILE TRUE DO
            IF DI_01 = 1 AND DI_02 = 0 THEN  !verificar que solo se presiono un botón
                TPWrite "Comenzando avance de la banda";
                Set Conveyor_INV;
                WaitTime 10.3;  !cambiar este para modificar tiempo de espera entre encendido y apagado
                Reset Conveyor_INV;
                TPWrite "Banda transportadora detenida";
                TPWrite "Iniciando Decoración del pastel";
                Set DO_01; ! bombillo que avisa del proceso de decoración
                MoveAbsJ RomperSingular, v1000, z1, Soporte_final;
                Path_10; ! Primero Ariadna
                TPWrite "Decoración ------> 34%";
                Path_20;
                TPWrite "Decoración ------> 67%";
                Path_30;
                TPWrite "Decoración ------> 100%";
                GoHome;
                WaitTime 2; !verificar este Gohome que hace.
                TPWrite "Comenzando avance de la banda";
                Set Conveyor_INV;
                WaitTime 3; ! si la caja se cae es por esto.
                Reset Conveyor_INV;
                TPWrite "Banda transportadora detenida";


            ELSEIF DI_01 = 0 AND DI_02=1 THEN
                TPWrite "Rutina de Mantenimiento empezando";
                Reset DO_01; ! apagando indicador de rutina de decoración
                Set DO_02; ! indicador de la rutina de mantenimiento
                GoHome;
                MoveAbsJ cambio_Tool, v300, z5, Soporte_final;
                TPWrite "CUIDADO OPERARIO CERCA AL ROBOT";
                TPWrite "Presione Boton1 y Boton2 al tiempo, para continuar";
                WaitUntil DI_01=1 AND DI_02=1;
                TPWrite "Continuando Programa...";
                WaitTime 6; ! tiempo de espera para asegurarse que el operario salio.
                MoveAbsJ HOME_Origen, v300, fine, Soporte_final;
                Reset DO_02;
            ELSEIF DI_01 = 0 AND DI_02=0 THEN
                TPWrite "Esperando Instrucciones";
                ! aqui iba un Waittime pero no pienso que sea neccesario
            ENDIF
             ! revisar si es necesario otro estado
        ENDWHILE


    ENDPROC

       PROC GoHome()
        CONST num tolerancia := 0.2;
        VAR jointtarget jt;
        jt := CJointT(); ! posición actual del robot
        IF  Abs(jt.robax.rax_1) < tolerancia AND
            Abs(jt.robax.rax_2) < tolerancia AND
            Abs(jt.robax.rax_3) < tolerancia AND
            Abs(jt.robax.rax_4) < tolerancia AND
            Abs(jt.robax.rax_5) < tolerancia AND
            Abs(jt.robax.rax_6) < tolerancia THEN
            TPWrite "Robot en home articular en 0°";
        ELSE
            TPWrite "Yendo a Home";

            MoveAbsJ HOME_Origen, v100, fine, Soporte_final;
            TPWrite "Robot en Home";
        ENDIF
    ENDPROC

    PROC Path_10()
        MoveJ Target_minihome,v100,z5,Soporte_final\WObj:=ADwob;
        MoveJ Target_200,v100,z5,Soporte_final\WObj:=ADwob;
        MoveL Target_210,v100,z5,Soporte_final\WObj:=ADwob;
        MoveL Target_220,v100,z5,Soporte_final\WObj:=ADwob;
        MoveL Target_230,v100,z5,Soporte_final\WObj:=ADwob;
        MoveL Target_240,v100,z5,Soporte_final\WObj:=ADwob;
        MoveL Target_250,v100,z5,Soporte_final\WObj:=ADwob;
        MoveL Target_260,v100,z5,Soporte_final\WObj:=ADwob;
        MoveL Target_270,v100,z5,Soporte_final\WObj:=ADwob;
        MoveL Target_280,v100,z5,Soporte_final\WObj:=ADwob;
        MoveL Target_210,v100,z5,Soporte_final\WObj:=ADwob;
        MoveL Target_200,v100,z5,Soporte_final\WObj:=ADwob;
        MoveL Target_290,v100,z5,Soporte_final\WObj:=ADwob;
        MoveL Target_300,v100,z5,Soporte_final\WObj:=ADwob;
        MoveL Target_310,v100,z5,Soporte_final\WObj:=ADwob;
        MoveL Target_320,v100,z5,Soporte_final\WObj:=ADwob;
        MoveL Target_300,v100,z5,Soporte_final\WObj:=ADwob;
        MoveL Target_290,v100,z5,Soporte_final\WObj:=ADwob;
        MoveL Target_330,v100,z5,Soporte_final\WObj:=ADwob;
        MoveL Target_340,v100,z5,Soporte_final\WObj:=ADwob;
        MoveL Target_350,v100,z5,Soporte_final\WObj:=ADwob;
        MoveL Target_360,v100,z5,Soporte_final\WObj:=ADwob;
        MoveL Target_370,v100,z5,Soporte_final\WObj:=ADwob;
        MoveL Target_380,v100,z5,Soporte_final\WObj:=ADwob;
        MoveL Target_390,v100,z5,Soporte_final\WObj:=ADwob;
        MoveL Target_400,v100,z5,Soporte_final\WObj:=ADwob;
        MoveL Target_410,v100,z5,Soporte_final\WObj:=ADwob;
        MoveL Target_420,v100,z5,Soporte_final\WObj:=ADwob;
        MoveL Target_430,v100,z5,Soporte_final\WObj:=ADwob;
        MoveL Target_440,v100,z5,Soporte_final\WObj:=ADwob;
        MoveL Target_340,v100,z5,Soporte_final\WObj:=ADwob;
        MoveL Target_330,v100,z5,Soporte_final\WObj:=ADwob;
        MoveL Target_450,v100,z5,Soporte_final\WObj:=ADwob;
        MoveL Target_460,v100,z5,Soporte_final\WObj:=ADwob;
        MoveL Target_470,v100,z5,Soporte_final\WObj:=ADwob;
        MoveL Target_480,v100,z5,Soporte_final\WObj:=ADwob;
        MoveL Target_490,v100,z5,Soporte_final\WObj:=ADwob;
        MoveL Target_460,v100,z5,Soporte_final\WObj:=ADwob;
        MoveL Target_450,v100,z5,Soporte_final\WObj:=ADwob;
        MoveL Target_500,v100,z5,Soporte_final\WObj:=ADwob;
        MoveL Target_510,v100,z5,Soporte_final\WObj:=ADwob;
        MoveL Target_520,v100,z5,Soporte_final\WObj:=ADwob;
        MoveL Target_530,v100,z5,Soporte_final\WObj:=ADwob;
        MoveL Target_540,v100,z5,Soporte_final\WObj:=ADwob;
        MoveL Target_550,v100,z5,Soporte_final\WObj:=ADwob;
        MoveL Target_560,v100,z5,Soporte_final\WObj:=ADwob;
        MoveL Target_570,v100,z5,Soporte_final\WObj:=ADwob;
        MoveL Target_580,v100,z5,Soporte_final\WObj:=ADwob;
        MoveL Target_590,v100,z5,Soporte_final\WObj:=ADwob;
        MoveL Target_500,v100,z5,Soporte_final\WObj:=ADwob;
        MoveL Target_600,v100,z5,Soporte_final\WObj:=ADwob;
        MoveL Target_610,v100,z5,Soporte_final\WObj:=ADwob; !baja en z letra 2 a
        MoveL Target_620,v100,z5,Soporte_final\WObj:=ADwob;
        MoveL Target_630,v100,z5,Soporte_final\WObj:=ADwob;
        MoveL Target_640,v100,z5,Soporte_final\WObj:=ADwob;
        MoveL Target_650,v100,z5,Soporte_final\WObj:=ADwob;
        MoveL Target_660,v100,z5,Soporte_final\WObj:=ADwob;
        MoveL Target_670,v100,z5,Soporte_final\WObj:=ADwob;
        MoveL Target_680,v100,z5,Soporte_final\WObj:=ADwob;
        MoveL Target_690,v100,z5,Soporte_final\WObj:=ADwob;
        MoveL Target_700,v100,z5,Soporte_final\WObj:=ADwob;
        MoveL Target_710,v100,z5,Soporte_final\WObj:=ADwob;
        MoveL Target_720,v100,z5,Soporte_final\WObj:=ADwob;
        MoveL Target_730,v100,z5,Soporte_final\WObj:=ADwob;
        MoveL Target_740,v100,z5,Soporte_final\WObj:=ADwob;
        MoveL Target_750,v100,z5,Soporte_final\WObj:=ADwob;
        MoveL Target_760,v100,z5,Soporte_final\WObj:=ADwob;
        MoveL Target_770,v100,z5,Soporte_final\WObj:=ADwob;
        MoveL Target_780,v100,z5,Soporte_final\WObj:=ADwob;
        MoveL Target_790,v100,z5,Soporte_final\WObj:=ADwob;
        MoveL Target_800,v100,z5,Soporte_final\WObj:=ADwob;
        MoveL Target_810,v100,z5,Soporte_final\WObj:=ADwob;
        MoveL Target_820,v100,z5,Soporte_final\WObj:=ADwob;
        MoveL Target_830,v100,z5,Soporte_final\WObj:=ADwob;
        MoveL Target_840,v100,z5,Soporte_final\WObj:=ADwob;
        MoveL Target_850,v100,z5,Soporte_final\WObj:=ADwob;
        MoveL Target_860,v100,z5,Soporte_final\WObj:=ADwob;
        MoveL Target_870,v100,z5,Soporte_final\WObj:=ADwob;
        MoveL Target_880,v100,z5,Soporte_final\WObj:=ADwob;
        MoveL Target_890,v100,z5,Soporte_final\WObj:=ADwob;
        MoveL Target_900,v100,z5,Soporte_final\WObj:=ADwob;
        MoveL Target_610,v100,z5,Soporte_final\WObj:=ADwob; !une las cosas en a
        MoveL Target_600,v100,z5,Soporte_final\WObj:=ADwob;
        MoveL Target_910,v100,z5,Soporte_final\WObj:=ADwob;
        MoveL Target_920,v100,z5,Soporte_final\WObj:=ADwob;
        MoveL Target_930,v100,z5,Soporte_final\WObj:=ADwob;
        MoveL Target_940,v100,z5,Soporte_final\WObj:=ADwob;
        MoveL Target_950,v100,z5,Soporte_final\WObj:=ADwob;
        MoveL Target_960,v100,z5,Soporte_final\WObj:=ADwob;
        MoveL Target_970,v100,z5,Soporte_final\WObj:=ADwob;
        MoveL Target_980,v100,z5,Soporte_final\WObj:=ADwob;
        MoveL Target_990,v100,z5,Soporte_final\WObj:=ADwob;
        MoveL Target_1000,v100,z5,Soporte_final\WObj:=ADwob;
        MoveL Target_1010,v100,z5,Soporte_final\WObj:=ADwob;
        MoveL Target_1020,v100,z5,Soporte_final\WObj:=ADwob;
        MoveL Target_1030,v100,z5,Soporte_final\WObj:=ADwob;
        MoveL Target_1040,v100,z5,Soporte_final\WObj:=ADwob;
        MoveL Target_1050,v100,z5,Soporte_final\WObj:=ADwob;
        MoveL Target_1060,v100,z5,Soporte_final\WObj:=ADwob;
        MoveL Target_1070,v100,z5,Soporte_final\WObj:=ADwob;
        MoveL Target_1080,v100,z5,Soporte_final\WObj:=ADwob;
        MoveL Target_1090,v100,z5,Soporte_final\WObj:=ADwob;
        MoveL Target_1100,v100,z5,Soporte_final\WObj:=ADwob;
        MoveL Target_920,v100,z5,Soporte_final\WObj:=ADwob;
        MoveL Target_910,v100,z5,Soporte_final\WObj:=ADwob;
        MoveL Target_1110,v100,z5,Soporte_final\WObj:=ADwob;
        MoveL Target_1120,v100,z5,Soporte_final\WObj:=ADwob;
        MoveL Target_1130,v100,z5,Soporte_final\WObj:=ADwob;
        MoveL Target_1140,v100,z5,Soporte_final\WObj:=ADwob;
        MoveL Target_1150,v100,z5,Soporte_final\WObj:=ADwob;
        MoveL Target_1160,v100,z5,Soporte_final\WObj:=ADwob;
        MoveL Target_1170,v100,z5,Soporte_final\WObj:=ADwob;
        MoveL Target_1180,v100,z5,Soporte_final\WObj:=ADwob;
        MoveL Target_1190,v100,z5,Soporte_final\WObj:=ADwob;
        MoveL Target_1200,v100,z5,Soporte_final\WObj:=ADwob;
        MoveL Target_1210,v100,z5,Soporte_final\WObj:=ADwob;
        MoveL Target_1220,v100,z5,Soporte_final\WObj:=ADwob;
        MoveL Target_1230,v100,z5,Soporte_final\WObj:=ADwob;
        MoveL Target_1240,v100,z5,Soporte_final\WObj:=ADwob;
        MoveL Target_1250,v100,z5,Soporte_final\WObj:=ADwob;
        MoveL Target_1260,v100,z5,Soporte_final\WObj:=ADwob;
        MoveL Target_1270,v100,z5,Soporte_final\WObj:=ADwob;
        MoveL Target_1280,v100,z5,Soporte_final\WObj:=ADwob;
        MoveL Target_1290,v100,z5,Soporte_final\WObj:=ADwob;
        MoveL Target_1300,v100,z5,Soporte_final\WObj:=ADwob;
        MoveL Target_1310,v100,z5,Soporte_final\WObj:=ADwob;
        MoveL Target_1320,v100,z5,Soporte_final\WObj:=ADwob;
        MoveL Target_1330,v100,z5,Soporte_final\WObj:=ADwob;
        MoveL Target_1340,v100,z5,Soporte_final\WObj:=ADwob;
        MoveL Target_1350,v100,z5,Soporte_final\WObj:=ADwob;
        MoveL Target_1360,v100,z5,Soporte_final\WObj:=ADwob;
        MoveL Target_1120,v100,z5,Soporte_final\WObj:=ADwob;
        MoveL Target_1110,v100,z5,Soporte_final\WObj:=ADwob;
        MoveL Target_1370,v100,z5,Soporte_final\WObj:=ADwob;
        MoveL Target_1380,v100,z5,Soporte_final\WObj:=ADwob;
        MoveL Target_1390,v100,z5,Soporte_final\WObj:=ADwob;
        MoveL Target_1400,v100,z5,Soporte_final\WObj:=ADwob;
        MoveL Target_1410,v100,z5,Soporte_final\WObj:=ADwob;
        MoveL Target_1420,v100,z5,Soporte_final\WObj:=ADwob;
        MoveL Target_1430,v100,z5,Soporte_final\WObj:=ADwob;
        MoveL Target_1440,v100,z5,Soporte_final\WObj:=ADwob;
        MoveL Target_1450,v100,z5,Soporte_final\WObj:=ADwob;
        MoveL Target_1460,v100,z5,Soporte_final\WObj:=ADwob;
        MoveL Target_1470,v100,z5,Soporte_final\WObj:=ADwob;
        MoveL Target_1480,v100,z5,Soporte_final\WObj:=ADwob;
        MoveL Target_1490,v100,z5,Soporte_final\WObj:=ADwob;
        MoveL Target_1500,v100,z5,Soporte_final\WObj:=ADwob;
        MoveL Target_1510,v100,z5,Soporte_final\WObj:=ADwob;
        MoveL Target_1520,v100,z5,Soporte_final\WObj:=ADwob;
        MoveL Target_1530,v100,z5,Soporte_final\WObj:=ADwob;
        MoveL Target_1540,v100,z5,Soporte_final\WObj:=ADwob;
        MoveL Target_1550,v100,z5,Soporte_final\WObj:=ADwob;
        MoveL Target_1560,v100,z5,Soporte_final\WObj:=ADwob;
        MoveL Target_1570,v100,z5,Soporte_final\WObj:=ADwob;
        MoveL Target_1580,v100,z5,Soporte_final\WObj:=ADwob;
        MoveL Target_1590,v100,z5,Soporte_final\WObj:=ADwob;
        MoveL Target_1600,v100,z5,Soporte_final\WObj:=ADwob;
        MoveL Target_1610,v100,z5,Soporte_final\WObj:=ADwob;
        MoveL Target_1620,v100,z5,Soporte_final\WObj:=ADwob;
        MoveL Target_1630,v100,z5,Soporte_final\WObj:=ADwob;
        MoveL Target_1640,v100,z5,Soporte_final\WObj:=ADwob;
        MoveL Target_1650,v100,z5,Soporte_final\WObj:=ADwob;
        MoveL Target_1660,v100,z5,Soporte_final\WObj:=ADwob;
        MoveL Target_1670,v100,z5,Soporte_final\WObj:=ADwob;
        MoveL Target_1680,v100,z5,Soporte_final\WObj:=ADwob;
        MoveL Target_1690,v100,z5,Soporte_final\WObj:=ADwob;
        MoveL Target_1700,v100,z5,Soporte_final\WObj:=ADwob;
        MoveL Target_1710,v100,z5,Soporte_final\WObj:=ADwob;
        MoveL Target_1720,v100,z5,Soporte_final\WObj:=ADwob;
        MoveL Target_1730,v100,z5,Soporte_final\WObj:=ADwob;
        MoveL Target_1740,v100,z5,Soporte_final\WObj:=ADwob;
        MoveL Target_1750,v100,z5,Soporte_final\WObj:=ADwob;
        MoveL Target_1760,v100,z5,Soporte_final\WObj:=ADwob;
        MoveL Target_1770,v100,z5,Soporte_final\WObj:=ADwob;
        MoveL Target_1780,v100,z5,Soporte_final\WObj:=ADwob;
        MoveL Target_1790,v100,z5,Soporte_final\WObj:=ADwob;
        MoveL Target_1800,v100,z5,Soporte_final\WObj:=ADwob;
        MoveL Target_1810,v100,z5,Soporte_final\WObj:=ADwob;
        MoveL Target_1820,v100,z5,Soporte_final\WObj:=ADwob;
        MoveL Target_1830,v100,z5,Soporte_final\WObj:=ADwob;
        MoveL Target_1840,v100,z5,Soporte_final\WObj:=ADwob;
        MoveL Target_1850,v100,z5,Soporte_final\WObj:=ADwob;
        MoveL Target_1860,v100,z5,Soporte_final\WObj:=ADwob;
        MoveL Target_1870,v100,z5,Soporte_final\WObj:=ADwob;
        MoveL Target_1880,v100,z5,Soporte_final\WObj:=ADwob;
        MoveL Target_1890,v100,z5,Soporte_final\WObj:=ADwob;
        MoveL Target_1900,v100,z5,Soporte_final\WObj:=ADwob;
        MoveL Target_1910,v100,z5,Soporte_final\WObj:=ADwob;
        MoveL Target_1920,v100,z5,Soporte_final\WObj:=ADwob;
        MoveL Target_1930,v100,z5,Soporte_final\WObj:=ADwob;
        MoveL Target_1940,v100,z5,Soporte_final\WObj:=ADwob;
        MoveL Target_1950,v100,z5,Soporte_final\WObj:=ADwob;
        MoveL Target_1960,v100,z5,Soporte_final\WObj:=ADwob;
        MoveL Target_1970,v100,z5,Soporte_final\WObj:=ADwob;
        MoveL Target_1980,v100,z5,Soporte_final\WObj:=ADwob;
        MoveL Target_1990,v100,z5,Soporte_final\WObj:=ADwob;
        MoveL Target_2000,v100,z5,Soporte_final\WObj:=ADwob;
        MoveL Target_2010,v100,z5,Soporte_final\WObj:=ADwob;
        MoveL Target_2020,v100,z5,Soporte_final\WObj:=ADwob;
        MoveL Target_2030,v100,z5,Soporte_final\WObj:=ADwob;
        MoveL Target_2040,v100,z5,Soporte_final\WObj:=ADwob;
        MoveL Target_2050,v100,z5,Soporte_final\WObj:=ADwob;
        MoveL Target_2060,v100,z5,Soporte_final\WObj:=ADwob;
        MoveL Target_2070,v100,z5,Soporte_final\WObj:=ADwob;
        MoveL Target_2080,v100,z5,Soporte_final\WObj:=ADwob;
        MoveL Target_2090,v100,z5,Soporte_final\WObj:=ADwob;
        MoveL Target_2100,v100,z5,Soporte_final\WObj:=ADwob;
        MoveL Target_2110,v100,z5,Soporte_final\WObj:=ADwob;
        MoveL Target_2120,v100,z5,Soporte_final\WObj:=ADwob;
        MoveL Target_2130,v100,z5,Soporte_final\WObj:=ADwob;
        MoveL Target_2140,v100,z5,Soporte_final\WObj:=ADwob;
        MoveL Target_2150,v100,z5,Soporte_final\WObj:=ADwob;
        MoveL Target_2160,v100,z5,Soporte_final\WObj:=ADwob;
        MoveL Target_2170,v100,z5,Soporte_final\WObj:=ADwob;
        MoveL Target_2180,v100,z5,Soporte_final\WObj:=ADwob;
        MoveL Target_2190,v100,z5,Soporte_final\WObj:=ADwob;
        MoveL Target_2200,v100,z5,Soporte_final\WObj:=ADwob;
        MoveL Target_2210,v100,z5,Soporte_final\WObj:=ADwob;
        MoveL Target_2220,v100,z5,Soporte_final\WObj:=ADwob;
        MoveL Target_2230,v100,z5,Soporte_final\WObj:=ADwob;
        MoveL Target_2240,v100,z5,Soporte_final\WObj:=ADwob;
        MoveL Target_1380,v100,z5,Soporte_final\WObj:=ADwob; !une letra a ultima
        MoveL Target_1370,v100,z5,Soporte_final\WObj:=ADwob; !sube en z
        MoveL Target_2250,v100,z5,Soporte_final\WObj:=ADwob; !circulos de las cosas
        MoveL Target_2260,v100,z5,Soporte_final\WObj:=ADwob;  !baja en z
        MoveL Target_2270,v100,z5,Soporte_final\WObj:=ADwob;
        MoveL Target_2280,v100,z5,Soporte_final\WObj:=ADwob;
        MoveL Target_2290,v100,z5,Soporte_final\WObj:=ADwob;
        MoveL Target_2300,v100,z5,Soporte_final\WObj:=ADwob;
        MoveL Target_2310,v100,z5,Soporte_final\WObj:=ADwob;
        MoveL Target_2320,v100,z5,Soporte_final\WObj:=ADwob;
        MoveL Target_2340,v100,z5,Soporte_final\WObj:=ADwob;
        MoveL Target_2350,v100,z5,Soporte_final\WObj:=ADwob;
        MoveL Target_2360,v100,z5,Soporte_final\WObj:=ADwob;
        MoveL Target_2370,v100,z5,Soporte_final\WObj:=ADwob;
        MoveL Target_2380,v100,z5,Soporte_final\WObj:=ADwob;
        MoveL Target_2390,v100,z5,Soporte_final\WObj:=ADwob;
        MoveL Target_2400,v100,z5,Soporte_final\WObj:=ADwob;
        MoveL Target_2410,v100,z5,Soporte_final\WObj:=ADwob;
        MoveL Target_2420,v100,z5,Soporte_final\WObj:=ADwob;
        MoveL Target_2430,v100,z5,Soporte_final\WObj:=ADwob;
        MoveL Target_2440,v100,z5,Soporte_final\WObj:=ADwob;
        MoveL Target_2450,v100,z5,Soporte_final\WObj:=ADwob;
        MoveL Target_2460,v100,z5,Soporte_final\WObj:=ADwob;
        MoveL Target_2470,v100,z5,Soporte_final\WObj:=ADwob;
        MoveL Target_2260,v100,z5,Soporte_final\WObj:=ADwob; !cierra circulo de a
        MoveL Target_2250,v100,z5,Soporte_final\WObj:=ADwob; !sube en z
        MoveL Target_2330,v100,z5,Soporte_final\WObj:=ADwob; !llega arriba en d
        MoveL Target_2500,v100,z5,Soporte_final\WObj:=ADwob;
        MoveL Target_2510,v100,z5,Soporte_final\WObj:=ADwob;
        MoveL Target_2520,v100,z5,Soporte_final\WObj:=ADwob;
        MoveL Target_2530,v100,z5,Soporte_final\WObj:=ADwob;
        MoveL Target_2540,v100,z5,Soporte_final\WObj:=ADwob;
        MoveL Target_2550,v100,z5,Soporte_final\WObj:=ADwob;
        MoveL Target_2560,v100,z5,Soporte_final\WObj:=ADwob;
        MoveL Target_2570,v100,z5,Soporte_final\WObj:=ADwob;
        MoveL Target_2580,v100,z5,Soporte_final\WObj:=ADwob;
        MoveL Target_2590,v100,z5,Soporte_final\WObj:=ADwob;
        MoveL Target_2600,v100,z5,Soporte_final\WObj:=ADwob;
        MoveL Target_2610,v100,z5,Soporte_final\WObj:=ADwob;
        MoveL Target_2620,v100,z5,Soporte_final\WObj:=ADwob;
        MoveL Target_2630,v100,z5,Soporte_final\WObj:=ADwob;
        MoveL Target_2640,v100,z5,Soporte_final\WObj:=ADwob;
        MoveL Target_2650,v100,z5,Soporte_final\WObj:=ADwob;
        MoveL Target_2660,v100,z5,Soporte_final\WObj:=ADwob;
        MoveL Target_2670,v100,z5,Soporte_final\WObj:=ADwob;
        MoveL Target_2690,v100,z5,Soporte_final\WObj:=ADwob;
        MoveL Target_2700,v100,z5,Soporte_final\WObj:=ADwob;
        MoveL Target_2710,v100,z5,Soporte_final\WObj:=ADwob;
        MoveL Target_2720,v100,z5,Soporte_final\WObj:=ADwob;
        MoveL Target_2730,v100,z5,Soporte_final\WObj:=ADwob;
        MoveL Target_2740,v100,z5,Soporte_final\WObj:=ADwob;
        MoveL Target_2750,v100,z5,Soporte_final\WObj:=ADwob;
        MoveL Target_2500,v100,z5,Soporte_final\WObj:=ADwob;
        MoveL Target_2330,v100,z5,Soporte_final\WObj:=ADwob;
        MoveL Target_2760,v100,z5,Soporte_final\WObj:=ADwob;
        MoveL Target_2770,v100,z5,Soporte_final\WObj:=ADwob;
        MoveL Target_2780,v100,z5,Soporte_final\WObj:=ADwob;
        MoveL Target_2790,v100,z5,Soporte_final\WObj:=ADwob;
        MoveL Target_2800,v100,z5,Soporte_final\WObj:=ADwob;
        MoveL Target_2810,v100,z5,Soporte_final\WObj:=ADwob;
        MoveL Target_2820,v100,z5,Soporte_final\WObj:=ADwob;
        MoveL Target_2830,v100,z5,Soporte_final\WObj:=ADwob;
        MoveL Target_2840,v100,z5,Soporte_final\WObj:=ADwob;
        MoveL Target_2850,v100,z5,Soporte_final\WObj:=ADwob;
        MoveL Target_2860,v100,z5,Soporte_final\WObj:=ADwob;
        MoveL Target_2870,v100,z5,Soporte_final\WObj:=ADwob;
        MoveL Target_2880,v100,z5,Soporte_final\WObj:=ADwob;
        MoveL Target_2890,v100,z5,Soporte_final\WObj:=ADwob;
        MoveL Target_2900,v100,z5,Soporte_final\WObj:=ADwob;
        MoveL Target_2910,v100,z5,Soporte_final\WObj:=ADwob;
        MoveL Target_2770,v100,z5,Soporte_final\WObj:=ADwob;
        MoveL Target_2760,v100,z5,Soporte_final\WObj:=ADwob; ! queda arriba final.
        MoveJ Target_minihome,v100,z5,Soporte_final\WObj:=ADwob;
    ENDPROC
    PROC Path_20()
        MoveJ Target_minihome,v100,z5,Soporte_final\WObj:=ADwob;
        MoveL Target_2920_up,v100,z5,Soporte_final\WObj:=ADwob;
        MoveL Target_2920,v100,z5,Soporte_final\WObj:=ADwob;
        MoveL Target_2930,v100,z5,Soporte_final\WObj:=ADwob;
        MoveC Target_2940,Target_2950,v100,z5,Soporte_final\WObj:=ADwob;
        MoveL Target_2960,v100,z5,Soporte_final\WObj:=ADwob;
                MoveL Target_2920,v100,z5,Soporte_final\WObj:=ADwob;
        MoveL Target_2970_up,v100,z5,Soporte_final\WObj:=ADwob;
        MoveL Target_2970,v100,z5,Soporte_final\WObj:=ADwob;
        MoveL Target_2980,v100,z5,Soporte_final\WObj:=ADwob;
        MoveC Target_2990,Target_3000,v100,z5,Soporte_final\WObj:=ADwob;
        MoveL Target_3010,v100,z5,Soporte_final\WObj:=ADwob;
                MoveL Target_2970,v100,z5,Soporte_final\WObj:=ADwob;
        MoveL Target_3030_2,v100,z5,Soporte_final\WObj:=ADwob;
        MoveL Target_3030,v100,z5,Soporte_final\WObj:=ADwob;
        MoveL Target_3040,v100,z5,Soporte_final\WObj:=ADwob;
        MoveL Target_3050,v100,z5,Soporte_final\WObj:=ADwob;
        MoveL Target_3060,v100,z5,Soporte_final\WObj:=ADwob;
        MoveL Target_3070,v100,z5,Soporte_final\WObj:=ADwob;
        MoveL Target_3080,v100,z5,Soporte_final\WObj:=ADwob;
        MoveL Target_3090,v100,z5,Soporte_final\WObj:=ADwob;
        MoveL Target_3100,v100,z5,Soporte_final\WObj:=ADwob;
        MoveL Target_3110,v100,z5,Soporte_final\WObj:=ADwob;
        MoveL Target_3120,v100,z5,Soporte_final\WObj:=ADwob;
        MoveL Target_3130,v100,z5,Soporte_final\WObj:=ADwob;
        MoveL Target_3140,v100,z5,Soporte_final\WObj:=ADwob;
        MoveL Target_3150,v100,z5,Soporte_final\WObj:=ADwob;
        MoveL Target_3160,v100,z5,Soporte_final\WObj:=ADwob;
        MoveL Target_3170,v100,z5,Soporte_final\WObj:=ADwob;
        MoveL Target_3180,v100,z5,Soporte_final\WObj:=ADwob;
        MoveL Target_3190,v100,z5,Soporte_final\WObj:=ADwob;
        MoveL Target_3200,v100,z5,Soporte_final\WObj:=ADwob;
        MoveL Target_3210,v100,z5,Soporte_final\WObj:=ADwob;
        MoveL Target_3220,v100,z5,Soporte_final\WObj:=ADwob;
        MoveL Target_3230,v100,z5,Soporte_final\WObj:=ADwob;
        MoveL Target_3240,v100,z5,Soporte_final\WObj:=ADwob;
        MoveL Target_3250,v100,z5,Soporte_final\WObj:=ADwob;
        MoveL Target_3030,v100,z5,Soporte_final\WObj:=ADwob;
        MoveL Target_3260_2,v100,z5,Soporte_final\WObj:=ADwob;
        MoveL Target_3260,v100,z5,Soporte_final\WObj:=ADwob;
        MoveL Target_3270,v100,z5,Soporte_final\WObj:=ADwob;
        MoveL Target_3280,v100,z5,Soporte_final\WObj:=ADwob;
        MoveL Target_3290,v100,z5,Soporte_final\WObj:=ADwob;
        MoveL Target_3300,v100,z5,Soporte_final\WObj:=ADwob;
        MoveL Target_3310,v100,z5,Soporte_final\WObj:=ADwob;
        MoveL Target_3320,v100,z5,Soporte_final\WObj:=ADwob;
        MoveL Target_3330,v100,z5,Soporte_final\WObj:=ADwob;
        MoveL Target_3340,v100,z5,Soporte_final\WObj:=ADwob;
        MoveL Target_3260,v100,z5,Soporte_final\WObj:=ADwob;
        MoveL Target_3350_2,v100,z5,Soporte_final\WObj:=ADwob;
        MoveL Target_3350,v100,z5,Soporte_final\WObj:=ADwob;
        MoveL Target_3360,v100,z5,Soporte_final\WObj:=ADwob;
        MoveL Target_3370,v100,z5,Soporte_final\WObj:=ADwob;
        MoveL Target_3380,v100,z5,Soporte_final\WObj:=ADwob;
        MoveL Target_3390,v100,z5,Soporte_final\WObj:=ADwob;
        MoveL Target_3400,v100,z5,Soporte_final\WObj:=ADwob;
        MoveL Target_3410,v100,z5,Soporte_final\WObj:=ADwob;
        MoveL Target_3350,v100,z5,Soporte_final\WObj:=ADwob;
        MoveL Target_3420_2,v100,z5,Soporte_final\WObj:=ADwob;
        MoveL Target_3420,v100,z5,Soporte_final\WObj:=ADwob;
        MoveL Target_3430,v100,z5,Soporte_final\WObj:=ADwob;
        MoveL Target_3440,v100,z5,Soporte_final\WObj:=ADwob;
        MoveL Target_3450,v100,z5,Soporte_final\WObj:=ADwob;
        MoveL Target_3420,v100,z5,Soporte_final\WObj:=ADwob;
        MoveL Target_3460_2,v100,z5,Soporte_final\WObj:=ADwob;
        MoveL Target_3460,v100,z5,Soporte_final\WObj:=ADwob;
        MoveL Target_3470,v100,z5,Soporte_final\WObj:=ADwob;
        MoveL Target_3480,v100,z5,Soporte_final\WObj:=ADwob;
        MoveL Target_3490,v100,z5,Soporte_final\WObj:=ADwob;
        MoveL Target_3500,v100,z5,Soporte_final\WObj:=ADwob;
        MoveL Target_3510,v100,z5,Soporte_final\WObj:=ADwob;
                MoveL Target_3460,v100,z5,Soporte_final\WObj:=ADwob;
                MoveL Target_3520_2,v100,z5,Soporte_final\WObj:=ADwob;
                MoveL Target_3520,v100,z5,Soporte_final\WObj:=ADwob;
        MoveL Target_3530,v100,z5,Soporte_final\WObj:=ADwob;
        MoveL Target_3540,v100,z5,Soporte_final\WObj:=ADwob;
        MoveL Target_3550,v100,z5,Soporte_final\WObj:=ADwob;
        MoveL Target_3560,v100,z5,Soporte_final\WObj:=ADwob;
        MoveL Target_3570,v100,z5,Soporte_final\WObj:=ADwob;
        MoveL Target_3580,v100,z5,Soporte_final\WObj:=ADwob;
                MoveL Target_3590,v100,z5,Soporte_final\WObj:=ADwob;
                MoveL Target_3600,v100,z5,Soporte_final\WObj:=ADwob;
        MoveL Target_3610,v100,z5,Soporte_final\WObj:=ADwob;
        MoveL Target_3620,v100,z5,Soporte_final\WObj:=ADwob;
        MoveL Target_3630,v100,z5,Soporte_final\WObj:=ADwob;
        MoveL Target_3640,v100,z5,Soporte_final\WObj:=ADwob;
        MoveL Target_3650,v100,z5,Soporte_final\WObj:=ADwob;
        MoveL Target_3660,v100,z5,Soporte_final\WObj:=ADwob;
        MoveL Target_3520,v100,z5,Soporte_final\WObj:=ADwob;
                MoveL Target_3670_2,v100,z5,Soporte_final\WObj:=ADwob;
                MoveL Target_3670,v100,z5,Soporte_final\WObj:=ADwob;
                MoveL Target_3680,v100,z5,Soporte_final\WObj:=ADwob;
        MoveL Target_3690,v100,z5,Soporte_final\WObj:=ADwob;
        MoveL Target_3700,v100,z5,Soporte_final\WObj:=ADwob;
        MoveL Target_3710,v100,z5,Soporte_final\WObj:=ADwob;
        MoveL Target_3720,v100,z5,Soporte_final\WObj:=ADwob;
        MoveL Target_3730,v100,z5,Soporte_final\WObj:=ADwob;
        MoveL Target_3740,v100,z5,Soporte_final\WObj:=ADwob;
        MoveL Target_3670,v100,z5,Soporte_final\WObj:=ADwob;
        MoveJ Target_minihome,v100,z5,Soporte_final\WObj:=ADwob;
    ENDPROC
    PROC Path_30()
                MoveL Target_3750_2,v100,z5,Soporte_final\WObj:=ADwob;
        MoveL Target_3750,v100,z5,Soporte_final\WObj:=ADwob;
        MoveL Target_3760,v100,z5,Soporte_final\WObj:=ADwob;
        MoveL Target_3770,v100,z5,Soporte_final\WObj:=ADwob;
        MoveL Target_3780,v100,z5,Soporte_final\WObj:=ADwob;
        MoveL Target_3790,v100,z5,Soporte_final\WObj:=ADwob;
        MoveL Target_3800,v100,z5,Soporte_final\WObj:=ADwob;
        MoveL Target_3810,v100,z5,Soporte_final\WObj:=ADwob;
        MoveL Target_3820,v100,z5,Soporte_final\WObj:=ADwob;
        MoveL Target_3830,v100,z5,Soporte_final\WObj:=ADwob;
        MoveL Target_3840,v100,z5,Soporte_final\WObj:=ADwob;
        MoveL Target_3850,v100,z5,Soporte_final\WObj:=ADwob;
        MoveL Target_3860,v100,z5,Soporte_final\WObj:=ADwob;
        MoveL Target_3870,v100,z5,Soporte_final\WObj:=ADwob;
        MoveL Target_3880,v100,z5,Soporte_final\WObj:=ADwob;
        MoveL Target_3890,v100,z5,Soporte_final\WObj:=ADwob;
        MoveL Target_3900,v100,z5,Soporte_final\WObj:=ADwob;
                MoveL Target_3750,v100,z5,Soporte_final\WObj:=ADwob;
                MoveL Target_3910_2,v100,z5,Soporte_final\WObj:=ADwob;
        MoveL Target_3910,v100,z5,Soporte_final\WObj:=ADwob;
        MoveL Target_3920,v100,z5,Soporte_final\WObj:=ADwob;
        MoveL Target_3930,v100,z5,Soporte_final\WObj:=ADwob;
        MoveL Target_3940,v100,z5,Soporte_final\WObj:=ADwob;
        MoveL Target_3950,v100,z5,Soporte_final\WObj:=ADwob;
        MoveL Target_3960,v100,z5,Soporte_final\WObj:=ADwob;
                MoveL Target_3910,v100,z5,Soporte_final\WObj:=ADwob;
                MoveL Target_3970_2,v100,z5,Soporte_final\WObj:=ADwob;
        MoveL Target_3970,v100,z5,Soporte_final\WObj:=ADwob;
        MoveL Target_3980,v100,z5,Soporte_final\WObj:=ADwob;
        MoveL Target_3990,v100,z5,Soporte_final\WObj:=ADwob;
        MoveL Target_4000,v100,z5,Soporte_final\WObj:=ADwob;
                MoveL Target_3970,v100,z5,Soporte_final\WObj:=ADwob;
                MoveL Target_4010_2,v100,z5,Soporte_final\WObj:=ADwob;
        MoveL Target_4010,v100,z5,Soporte_final\WObj:=ADwob;
        MoveL Target_4020,v100,z5,Soporte_final\WObj:=ADwob;
        MoveL Target_4030,v100,z5,Soporte_final\WObj:=ADwob;
        MoveL Target_4040,v100,z5,Soporte_final\WObj:=ADwob;
        MoveL Target_4050,v100,z5,Soporte_final\WObj:=ADwob;
        MoveL Target_4060,v100,z5,Soporte_final\WObj:=ADwob;
        MoveL Target_4070,v100,z5,Soporte_final\WObj:=ADwob;
        MoveL Target_4080,v100,z5,Soporte_final\WObj:=ADwob;
        MoveL Target_4090,v100,z5,Soporte_final\WObj:=ADwob;
        MoveL Target_4100,v100,z5,Soporte_final\WObj:=ADwob;
        MoveL Target_4110,v100,z5,Soporte_final\WObj:=ADwob;
        MoveL Target_4120,v100,z5,Soporte_final\WObj:=ADwob;
        MoveL Target_4130,v100,z5,Soporte_final\WObj:=ADwob;
        MoveL Target_4010,v100,z5,Soporte_final\WObj:=ADwob;
        MoveL Target_minihome,v100,z5,Soporte_final\WObj:=ADwob;
    ENDPROC
ENDMODULE

--- Controller Data/IRB140_6_81/SYSPAR/EIO.cfg ---
EIO:CFG_1.0:6:1::
#
EIO_SIGNAL:

      -Name "DI_01" -SignalType "DI"

      -Name "DI_02" -SignalType "DI"

      -Name "Conveyor_INV" -SignalType "DO"

      -Name "Conveyor_FWD" -SignalType "DO"

      -Name "DO_01" -SignalType "DO"

      -Name "DO_02" -SignalType "DO"
